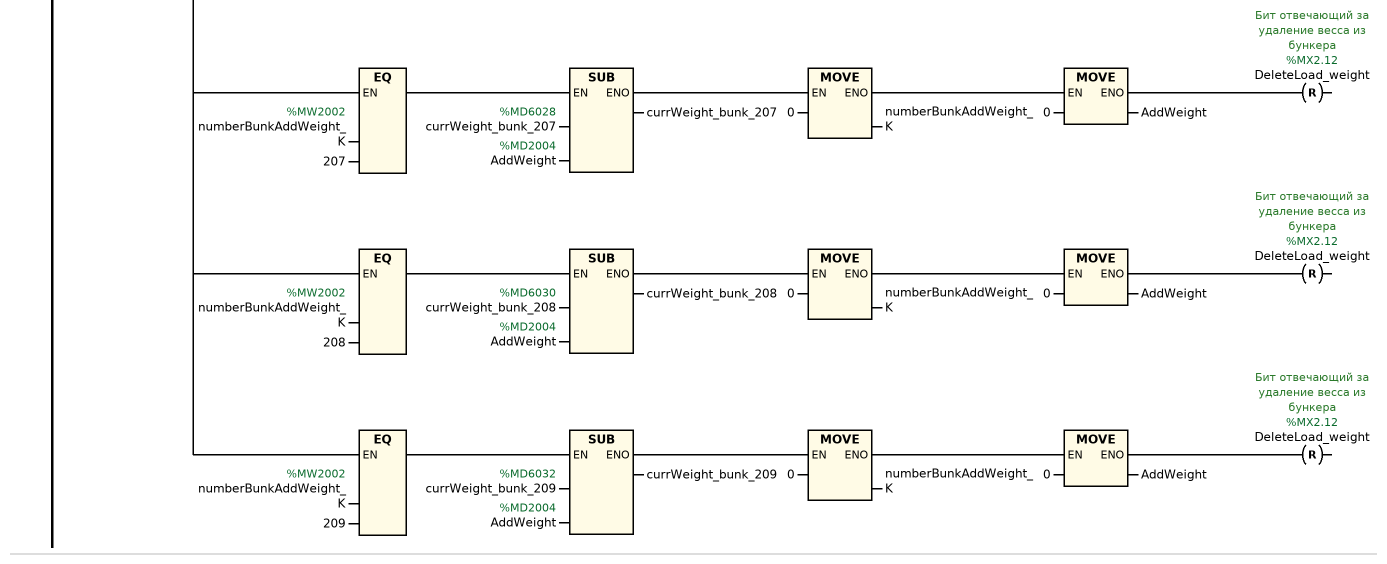
// NETWORK 2
//   DeleteLoad_weight: Бит отвечающий за удаление весса из бункера | AT %MX2.12
//   numberBunkAddWeight_Z: Храниться номер бункера для дабавления или удаления значения текущего весса в ручную... Сырье | AT %MW2000
//   currWeight_bunk_101: ----------------------------------------------------------------------------------------------------- текущий вес в зерновых бункерах ----------------------------------------------------------------------------------------------------- | AT %MD6000
//   AddWeight: Значение дабавляемого весса в бункер | AT %MD2004
//   currWeight_bunk_102: AT %MD6002
//   currWeight_bunk_103: AT %MD6004
//   currWeight_bunk_104: AT %MD6006
//   currWeight_bunk_105: AT %MD6008
//   currWeight_bunk_106: AT %MD6010
//   currWeight_bunk_107: AT %MD6012
//   currWeight_bunk_108: AT %MD6014
//   numberBunkAddWeight_K: Храниться номер бункера для дабавления или удаления значения текущего весса в ручную... Добавки | AT %MW2002
//   currWeight_bunk_201: ----------------------------------------------------------------------------------------------------- ----------------------------------------------------------------------------------------------------- текущий вес в бункерах компонентов ----------------------------------------------------------------------------------------------------- | AT %MD6016
//   currWeight_bunk_202: AT %MD6018
//   currWeight_bunk_203: AT %MD6020
//   currWeight_bunk_204: AT %MD6022
//   currWeight_bunk_205: AT %MD6024
//   currWeight_bunk_206: AT %MD6026
//   currWeight_bunk_207: AT %MD6028
//   currWeight_bunk_208: AT %MD6030
//   currWeight_bunk_209: AT %MD6032
_w2 := DeleteLoad_weight;
IF _w2 AND numberBunkAddWeight_Z = 101 THEN currWeight_bunk_101 := currWeight_bunk_101 - AddWeight; END_IF
IF _w2 AND numberBunkAddWeight_Z = 101 THEN numberBunkAddWeight_Z := 0; END_IF
IF _w2 AND numberBunkAddWeight_Z = 101 THEN AddWeight := 0; END_IF
DeleteLoad_weight R= _w2 AND numberBunkAddWeight_Z = 101;
IF _w2 AND numberBunkAddWeight_Z = 102 THEN currWeight_bunk_102 := currWeight_bunk_102 - AddWeight; END_IF
IF _w2 AND numberBunkAddWeight_Z = 102 THEN numberBunkAddWeight_Z := 0; END_IF
IF _w2 AND numberBunkAddWeight_Z = 102 THEN AddWeight := 0; END_IF
DeleteLoad_weight R= _w2 AND numberBunkAddWeight_Z = 102;
IF _w2 AND numberBunkAddWeight_Z = 103 THEN currWeight_bunk_103 := currWeight_bunk_103 - AddWeight; END_IF
IF _w2 AND numberBunkAddWeight_Z = 103 THEN numberBunkAddWeight_Z := 0; END_IF
IF _w2 AND numberBunkAddWeight_Z = 103 THEN AddWeight := 0; END_IF
DeleteLoad_weight R= _w2 AND numberBunkAddWeight_Z = 103;
IF _w2 AND numberBunkAddWeight_Z = 104 THEN currWeight_bunk_104 := currWeight_bunk_104 - AddWeight; END_IF
IF _w2 AND numberBunkAddWeight_Z = 104 THEN numberBunkAddWeight_Z := 0; END_IF
IF _w2 AND numberBunkAddWeight_Z = 104 THEN AddWeight := 0; END_IF
DeleteLoad_weight R= _w2 AND numberBunkAddWeight_Z = 104;
IF _w2 AND numberBunkAddWeight_Z = 105 THEN currWeight_bunk_105 := currWeight_bunk_105 - AddWeight; END_IF
IF _w2 AND numberBunkAddWeight_Z = 105 THEN numberBunkAddWeight_Z := 0; END_IF
IF _w2 AND numberBunkAddWeight_Z = 105 THEN AddWeight := 0; END_IF
DeleteLoad_weight R= _w2 AND numberBunkAddWeight_Z = 105;
IF _w2 AND numberBunkAddWeight_Z = 106 THEN currWeight_bunk_106 := currWeight_bunk_106 - AddWeight; END_IF
IF _w2 AND numberBunkAddWeight_Z = 106 THEN numberBunkAddWeight_Z := 0; END_IF
IF _w2 AND numberBunkAddWeight_Z = 106 THEN AddWeight := 0; END_IF
DeleteLoad_weight R= _w2 AND numberBunkAddWeight_Z = 106;
IF _w2 AND numberBunkAddWeight_Z = 107 THEN currWeight_bunk_107 := currWeight_bunk_107 - AddWeight; END_IF
IF _w2 AND numberBunkAddWeight_Z = 107 THEN numberBunkAddWeight_Z := 0; END_IF
IF _w2 AND numberBunkAddWeight_Z = 107 THEN AddWeight := 0; END_IF
DeleteLoad_weight R= _w2 AND numberBunkAddWeight_Z = 107;
IF _w2 AND numberBunkAddWeight_Z = 108 THEN currWeight_bunk_108 := currWeight_bunk_108 - AddWeight; END_IF
IF _w2 AND numberBunkAddWeight_Z = 108 THEN numberBunkAddWeight_Z := 0; END_IF
IF _w2 AND numberBunkAddWeight_Z = 108 THEN AddWeight := 0; END_IF
DeleteLoad_weight R= _w2 AND numberBunkAddWeight_Z = 108;
IF _w2 AND numberBunkAddWeight_K = 201 THEN currWeight_bunk_201 := currWeight_bunk_201 - AddWeight; END_IF
IF _w2 AND numberBunkAddWeight_K = 201 THEN numberBunkAddWeight_K := 0; END_IF
IF _w2 AND numberBunkAddWeight_K = 201 THEN AddWeight := 0; END_IF
DeleteLoad_weight R= _w2 AND numberBunkAddWeight_K = 201;
IF _w2 AND numberBunkAddWeight_K = 202 THEN currWeight_bunk_202 := currWeight_bunk_202 - AddWeight; END_IF
IF _w2 AND numberBunkAddWeight_K = 202 THEN numberBunkAddWeight_K := 0; END_IF
IF _w2 AND numberBunkAddWeight_K = 202 THEN AddWeight := 0; END_IF
DeleteLoad_weight R= _w2 AND numberBunkAddWeight_K = 202;
IF _w2 AND numberBunkAddWeight_K = 203 THEN currWeight_bunk_203 := currWeight_bunk_203 - AddWeight; END_IF
IF _w2 AND numberBunkAddWeight_K = 203 THEN numberBunkAddWeight_K := 0; END_IF
IF _w2 AND numberBunkAddWeight_K = 203 THEN AddWeight := 0; END_IF
DeleteLoad_weight R= _w2 AND numberBunkAddWeight_K = 203;
IF _w2 AND numberBunkAddWeight_K = 204 THEN currWeight_bunk_204 := currWeight_bunk_204 - AddWeight; END_IF
IF _w2 AND numberBunkAddWeight_K = 204 THEN numberBunkAddWeight_K := 0; END_IF
IF _w2 AND numberBunkAddWeight_K = 204 THEN AddWeight := 0; END_IF
DeleteLoad_weight R= _w2 AND numberBunkAddWeight_K = 204;
IF _w2 AND numberBunkAddWeight_K = 205 THEN currWeight_bunk_205 := currWeight_bunk_205 - AddWeight; END_IF
IF _w2 AND numberBunkAddWeight_K = 205 THEN numberBunkAddWeight_K := 0; END_IF
IF _w2 AND numberBunkAddWeight_K = 205 THEN AddWeight := 0; END_IF
DeleteLoad_weight R= _w2 AND numberBunkAddWeight_K = 205;
IF _w2 AND numberBunkAddWeight_K = 206 THEN currWeight_bunk_206 := currWeight_bunk_206 - AddWeight; END_IF
IF _w2 AND numberBunkAddWeight_K = 206 THEN numberBunkAddWeight_K := 0; END_IF
IF _w2 AND numberBunkAddWeight_K = 206 THEN AddWeight := 0; END_IF
DeleteLoad_weight R= _w2 AND numberBunkAddWeight_K = 206;
IF _w2 AND numberBunkAddWeight_K = 207 THEN currWeight_bunk_207 := currWeight_bunk_207 - AddWeight; END_IF
IF _w2 AND numberBunkAddWeight_K = 207 THEN numberBunkAddWeight_K := 0; END_IF
IF _w2 AND numberBunkAddWeight_K = 207 THEN AddWeight := 0; END_IF
DeleteLoad_weight R= _w2 AND numberBunkAddWeight_K = 207;
IF _w2 AND numberBunkAddWeight_K = 208 THEN currWeight_bunk_208 := currWeight_bunk_208 - AddWeight; END_IF
IF _w2 AND numberBunkAddWeight_K = 208 THEN numberBunkAddWeight_K := 0; END_IF
IF _w2 AND numberBunkAddWeight_K = 208 THEN AddWeight := 0; END_IF
DeleteLoad_weight R= _w2 AND numberBunkAddWeight_K = 208;
IF _w2 AND numberBunkAddWeight_K = 209 THEN currWeight_bunk_209 := currWeight_bunk_209 - AddWeight; END_IF
IF _w2 AND numberBunkAddWeight_K = 209 THEN numberBunkAddWeight_K := 0; END_IF
IF _w2 AND numberBunkAddWeight_K = 209 THEN AddWeight := 0; END_IF
DeleteLoad_weight R= _w2 AND numberBunkAddWeight_K = 209;

END_PROGRAM

// PLC_241/Application/CONVERT_REAL_TO_INT
PROGRAM CONVERT_REAL_TO_INT
VAR
END_VAR

								
								// Значение (процент компонента в рецепте)
	KP_101:= (INT_TO_REAL(iKP_101)/10.0);
	KP_102:= (INT_TO_REAL(iKP_102)/10.0);
	KP_103:= (INT_TO_REAL(iKP_103)/10.0);
	KP_104:= (INT_TO_REAL(iKP_104)/10.0);
	KP_105:= (INT_TO_REAL(iKP_105)/10.0);
	KP_106:= (INT_TO_REAL(iKP_106)/10.0);
	KP_107:= (INT_TO_REAL(iKP_107)/10.0);
	KP_108:= (INT_TO_REAL(iKP_108)/10.0);
	
								// Значение в кг, масса компонента в рецепте
	iK_101:= REAL_TO_INT(K_101*10.0);
	iK_102:= REAL_TO_INT(K_102*10.0);
	iK_103:= REAL_TO_INT(K_103*10.0);
	iK_104:= REAL_TO_INT(K_104*10.0);
	iK_105:= REAL_TO_INT(K_105*10.0);
	iK_106:= REAL_TO_INT(K_106*10.0);
	iK_107:= REAL_TO_INT(K_107*10.0);
	iK_108:= REAL_TO_INT(K_108*10.0);
	
								// Значение выбега 
	FALL_101:= (INT_TO_REAL(iFALL_101)/10.0);
	FALL_102:= (INT_TO_REAL(iFALL_102)/10.0);
	FALL_103:= (INT_TO_REAL(iFALL_103)/10.0);
	FALL_104:= (INT_TO_REAL(iFALL_104)/10.0);
	FALL_105:= (INT_TO_REAL(iFALL_105)/10.0);
	FALL_106:= (INT_TO_REAL(iFALL_106)/10.0);
	FALL_107:= (INT_TO_REAL(iFALL_107)/10.0);
	FALL_108:= (INT_TO_REAL(iFALL_108)/10.0);
	
								// Значение (Кг) при котором дазатор начинает снижать скорость дозирования для точного дозирования на весы
	vlDropSpeed_101:= (INT_TO_REAL(ivlDropSpeed_101)/10.0);
	vlDropSpeed_102:= (INT_TO_REAL(ivlDropSpeed_102)/10.0);
	vlDropSpeed_103:= (INT_TO_REAL(ivlDropSpeed_103)/10.0);
	vlDropSpeed_104:= (INT_TO_REAL(ivlDropSpeed_104)/10.0);
	vlDropSpeed_105:= (INT_TO_REAL(ivlDropSpeed_105)/10.0);
	vlDropSpeed_106:= (INT_TO_REAL(ivlDropSpeed_106)/10.0);
	vlDropSpeed_107:= (INT_TO_REAL(ivlDropSpeed_107)/10.0);
	vlDropSpeed_108:= (INT_TO_REAL(ivlDropSpeed_108)/10.0);
	
								// Значение (Кг) после автоматической коррекции падающег остоба (Выбега)
	iNewFall_101:= REAL_TO_INT(NewFall_101*10.0);
	iNewFall_102:= REAL_TO_INT(NewFall_102*10.0);
	iNewFall_103:= REAL_TO_INT(NewFall_103*10.0);
	iNewFall_104:= REAL_TO_INT(NewFall_104*10.0);
	iNewFall_105:= REAL_TO_INT(NewFall_105*10.0);
	iNewFall_106:= REAL_TO_INT(NewFall_106*10.0);
	iNewFall_107:= REAL_TO_INT(NewFall_107*10.0);
	iNewFall_108:= REAL_TO_INT(NewFall_108*10.0);

END_PROGRAM

// PLC_241/Application/POU/prgDOSING_BIG_WEIGHT
PROGRAM prgDOSING_BIG_WEIGHT
VAR
	Dozator_101: Dozator;
	T_20110: T;
	TON_pch_11_16: TON;
	
	vesi_big_done: BOOL;	// Вес сдозирован на весы
	Dozator_102: Dozator;
	Dozator_103: Dozator;
	Dozator_104: Dozator;
	Dozator_105: Dozator;
	Dozator_106: Dozator;
	TON_pch_17_18: TON;
	Dozator_107: Dozator;
	Dozator_108: Dozator;
	vesi_big_unldone: BOOL;
	TP_TARE_BIG: TP;
	CTU_BIG_WEIGHT: CTU;
END_VAR
VAR // added by the converter: edge detectors and wires of the graphical bodies
    _rt1, _rt2, _rt3, _rt4, _rt5, _rt6, _rt7, _rt8, _rt9, _rt10, _rt11 : R_TRIG;
    _ft1 : F_TRIG;
    _w1, _w2, _w3, _w4, _w5, _w6, _w7, _w8, _w9 : BOOL;
END_VAR

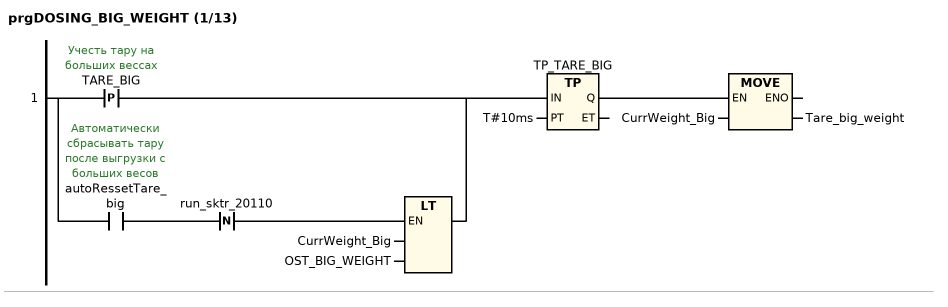
// NETWORK 1
//   TARE_BIG: Учесть тару на больших вессах
//   autoRessetTare_big: Автоматически сбрасывать тару после выгрузки с больших весов
//   CurrWeight_Big: Вес на больших весах
//   OST_BIG_WEIGHT: Остаток на больших весах (вводиться со скады)
//   Tare_big_weight: Вес тары на больших весах
_rt1(CLK := TARE_BIG);
_ft1(CLK := run_sktr_20110);
TP_TARE_BIG(IN := _rt1.Q OR autoRessetTare_big AND _ft1.Q AND CurrWeight_Big < OST_BIG_WEIGHT, PT := T#10ms); // TP
IF TP_TARE_BIG.Q THEN Tare_big_weight := CurrWeight_Big; END_IF

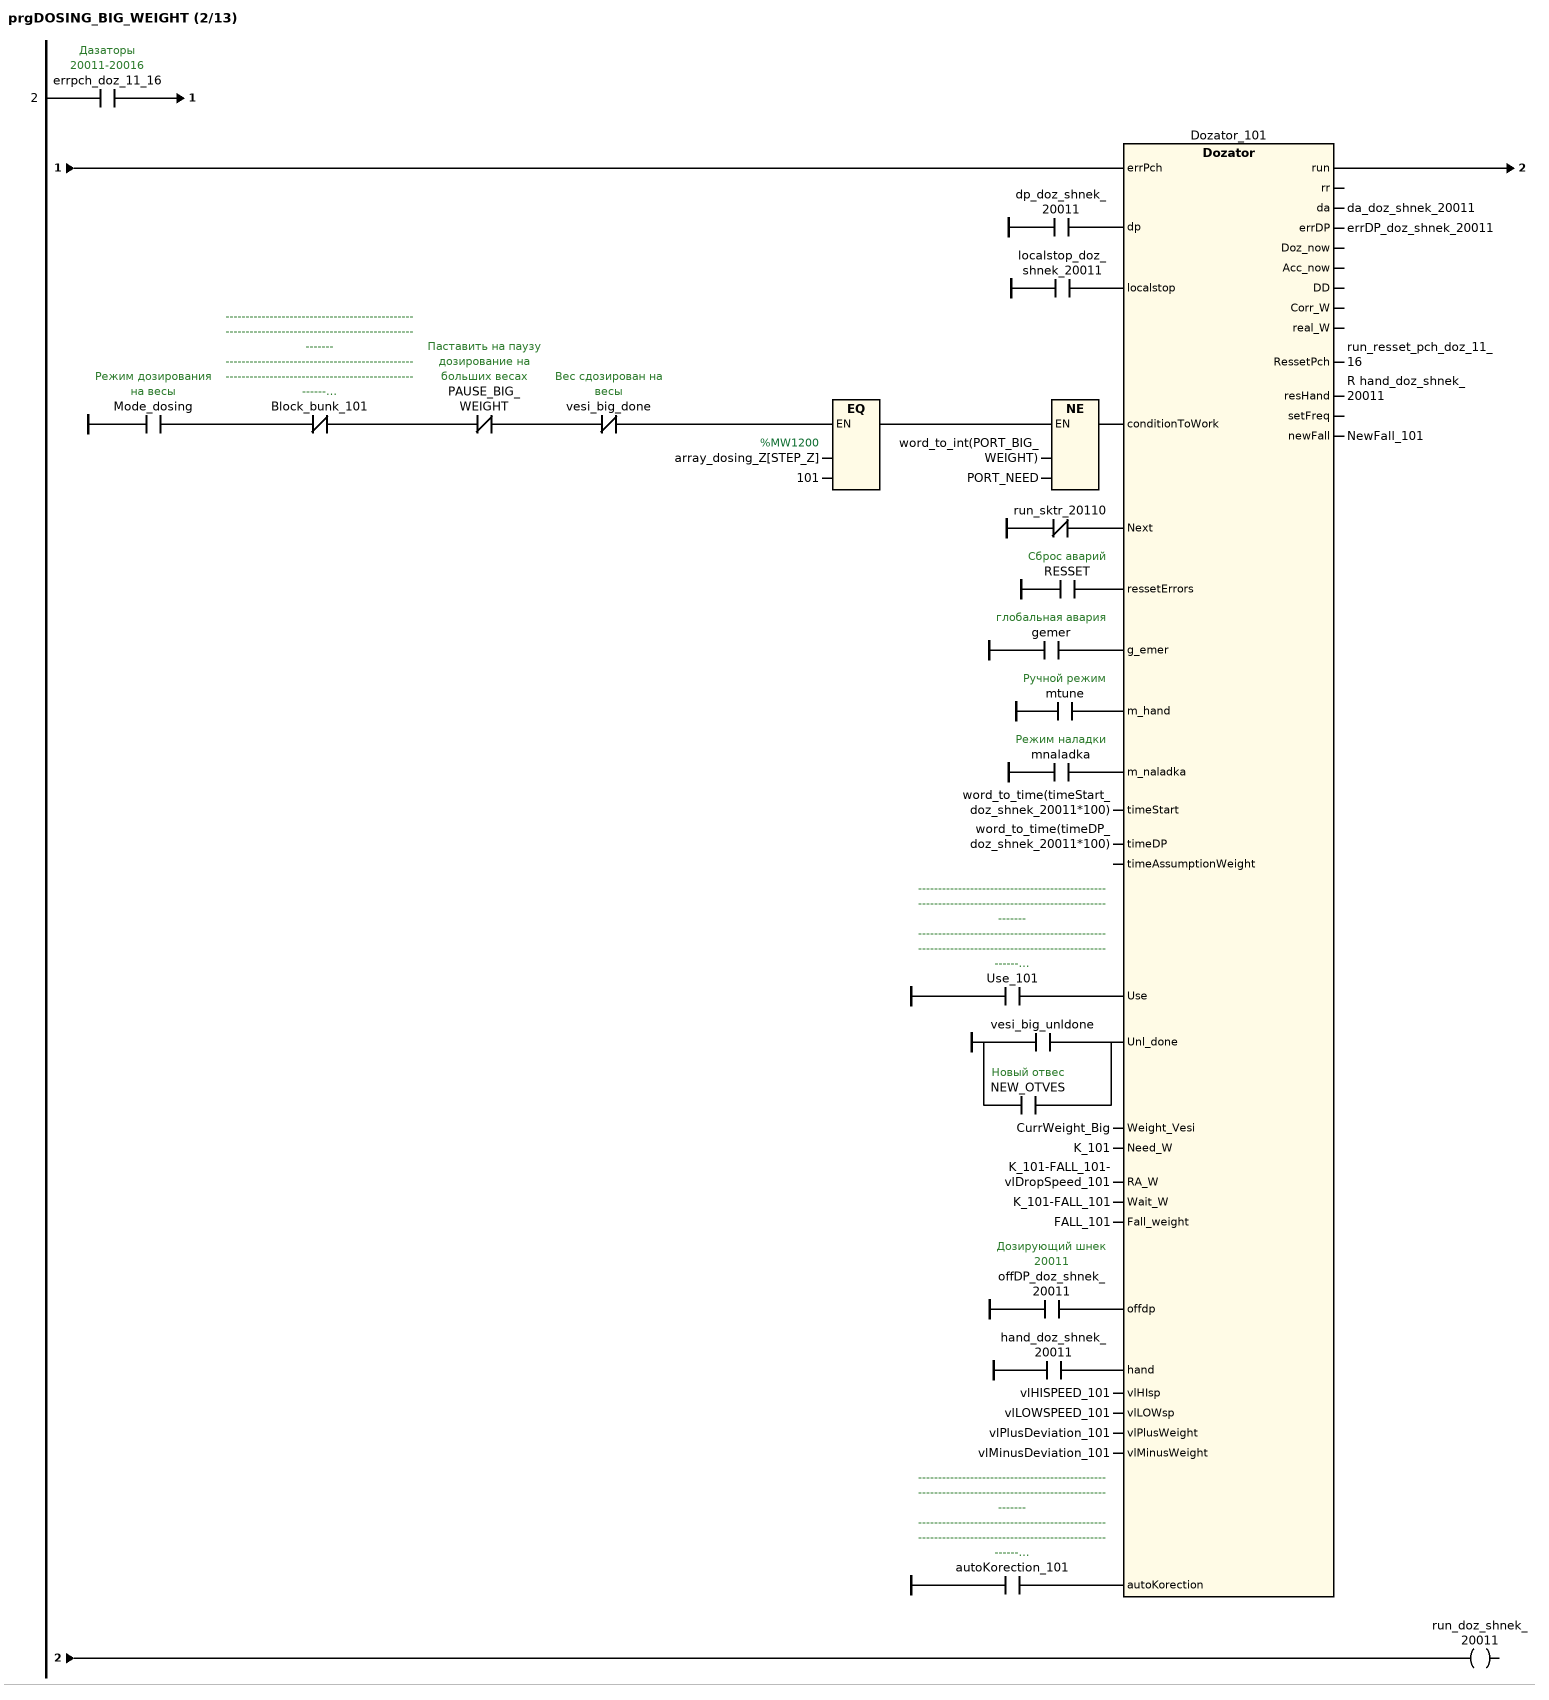
// NETWORK 2
//   errpch_doz_11_16: Дазаторы 20011-20016
//   Mode_dosing: Режим дозирования на весы
//   Block_bunk_101: ----------------------------------------------------------------------------------------------------- ----------------------------------------------------------------------------------------------------- Блокировка компонента на дозирование в рецепте -----------------------------------------------------------------------------------------------------
//   PAUSE_BIG_WEIGHT: Паставить на паузу дозирование на больших весах
//   vesi_big_done: Вес сдозирован на весы
//   array_dosing_Z[STEP_Z]: Массив очереди дозирования больших весов (в ячейке храниться номер бункера из которого нужно дозировать) | AT %MW1200
//   PORT_NEED: количество нужных порций
//   RESSET: Сброс аварий
//   gemer: глобальная авария
//   mtune: Ручной режим
//   mnaladka: Режим наладки
//   Use_101: ----------------------------------------------------------------------------------------------------- ----------------------------------------------------------------------------------------------------- Использование Дозатора в рецепте -----------------------------------------------------------------------------------------------------
//   NEW_OTVES: Новый отвес
//   CurrWeight_Big: Вес на больших весах
//   K_101: Значение реал для обработки контроллером
//   K_101-FALL_101-vlDropSpeed_101: Значение реал для обработки контроллером
//   K_101-FALL_101: Значение реал для обработки контроллером
//   FALL_101: Преобразованное значение падающего столба для обработки контроллером
//   offDP_doz_shnek_20011: Дозирующий шнек 20011
//   vlHISPEED_101: ----------------------------------------------------------------------------------------------------- ----------------------------------------------------------------------------------------------------- Значение (Гц) минимальной и максимальной скорости дозирования -----------------------------------------------------------------------------------------------------
//   vlPlusDeviation_101: ----------------------------------------------------------------------------------------------------- Значение (кг) допустимое отклонение +/- каждого компонента -----------------------------------------------------------------------------------------------------
//   autoKorection_101: ----------------------------------------------------------------------------------------------------- ----------------------------------------------------------------------------------------------------- Биты отвечающик за автоматический расчет падающего столба (Выбега) -----------------------------------------------------------------------------------------------------
//   errDP_doz_shnek_20011: Шнек Дозатор 20011
Dozator_101(
    errPch := errpch_doz_11_16,
    dp := dp_doz_shnek_20011,
    localstop := localstop_doz_shnek_20011,
    conditionToWork := Mode_dosing AND NOT Block_bunk_101 AND NOT PAUSE_BIG_WEIGHT AND NOT vesi_big_done AND array_dosing_Z[STEP_Z] = 101 AND (word_to_int(PORT_BIG_WEIGHT)) <> PORT_NEED,
    Next := NOT run_sktr_20110,
    ressetErrors := RESSET,
    g_emer := gemer,
    m_hand := mtune,
    m_naladka := mnaladka,
    timeStart := word_to_time(timeStart_doz_shnek_20011*100),
    timeDP := word_to_time(timeDP_doz_shnek_20011*100),
    Use := Use_101,
    Unl_done := vesi_big_unldone OR NEW_OTVES,
    Weight_Vesi := CurrWeight_Big,
    Need_W := K_101,
    RA_W := K_101-FALL_101-vlDropSpeed_101,
    Wait_W := K_101-FALL_101,
    Fall_weight := FALL_101,
    offdp := offDP_doz_shnek_20011,
    hand := hand_doz_shnek_20011,
    vlHIsp := vlHISPEED_101,
    vlLOWsp := vlLOWSPEED_101,
    vlPlusWeight := vlPlusDeviation_101,
    vlMinusWeight := vlMinusDeviation_101,
    autoKorection := autoKorection_101,
    da => da_doz_shnek_20011,
    errDP => errDP_doz_shnek_20011,
    RessetPch => run_resset_pch_doz_11_16,
    newFall => NewFall_101); // Dozator
hand_doz_shnek_20011 R= Dozator_101.resHand;
run_doz_shnek_20011 := Dozator_101.run;

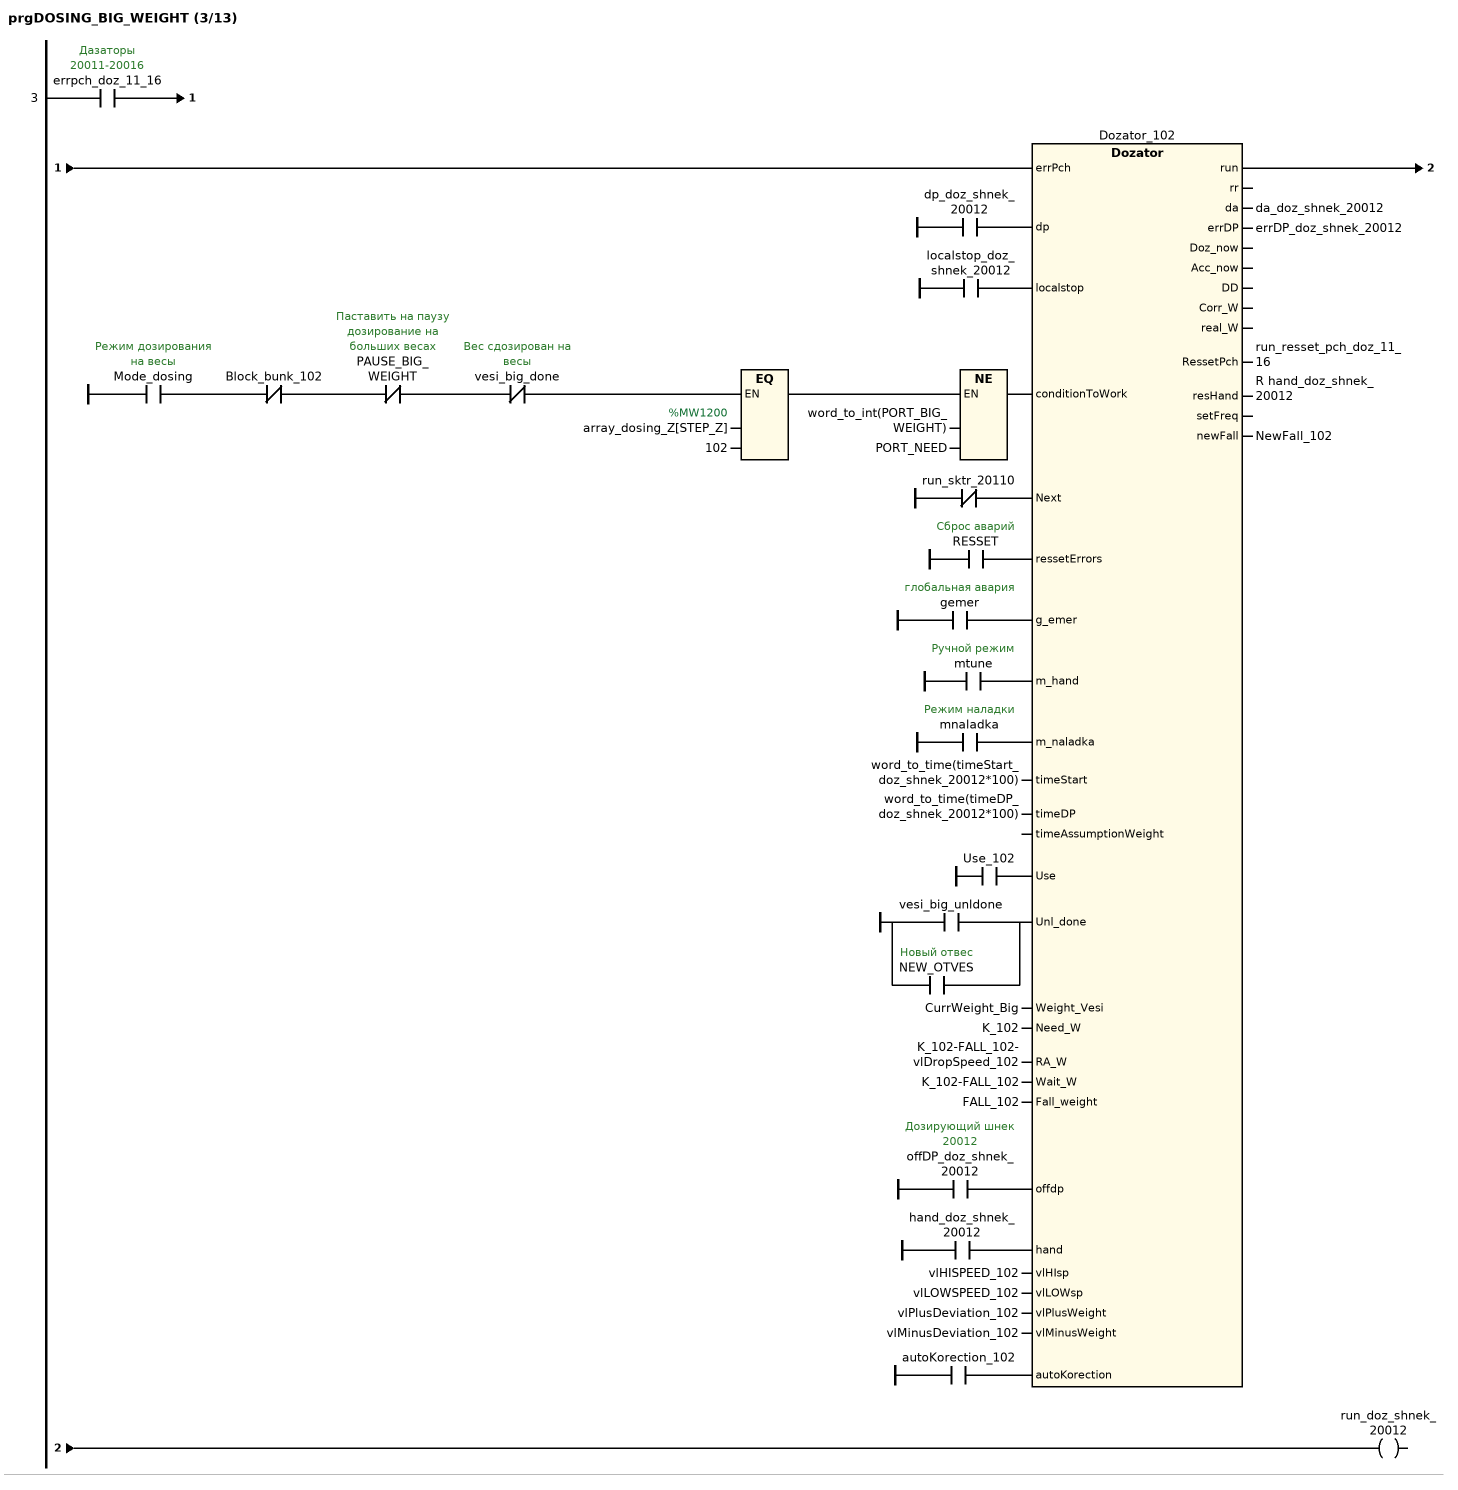
// NETWORK 3
//   errpch_doz_11_16: Дазаторы 20011-20016
//   Mode_dosing: Режим дозирования на весы
//   PAUSE_BIG_WEIGHT: Паставить на паузу дозирование на больших весах
//   vesi_big_done: Вес сдозирован на весы
//   array_dosing_Z[STEP_Z]: Массив очереди дозирования больших весов (в ячейке храниться номер бункера из которого нужно дозировать) | AT %MW1200
//   PORT_NEED: количество нужных порций
//   RESSET: Сброс аварий
//   gemer: глобальная авария
//   mtune: Ручной режим
//   mnaladka: Режим наладки
//   NEW_OTVES: Новый отвес
//   CurrWeight_Big: Вес на больших весах
//   offDP_doz_shnek_20012: Дозирующий шнек 20012
//   errDP_doz_shnek_20012: Шнек Дозатор 20012
Dozator_102(
    errPch := errpch_doz_11_16,
    dp := dp_doz_shnek_20012,
    localstop := localstop_doz_shnek_20012,
    conditionToWork := Mode_dosing AND NOT Block_bunk_102 AND NOT PAUSE_BIG_WEIGHT AND NOT vesi_big_done AND array_dosing_Z[STEP_Z] = 102 AND (word_to_int(PORT_BIG_WEIGHT)) <> PORT_NEED,
    Next := NOT run_sktr_20110,
    ressetErrors := RESSET,
    g_emer := gemer,
    m_hand := mtune,
    m_naladka := mnaladka,
    timeStart := word_to_time(timeStart_doz_shnek_20012*100),
    timeDP := word_to_time(timeDP_doz_shnek_20012*100),
    Use := Use_102,
    Unl_done := vesi_big_unldone OR NEW_OTVES,
    Weight_Vesi := CurrWeight_Big,
    Need_W := K_102,
    RA_W := K_102-FALL_102-vlDropSpeed_102,
    Wait_W := K_102-FALL_102,
    Fall_weight := FALL_102,
    offdp := offDP_doz_shnek_20012,
    hand := hand_doz_shnek_20012,
    vlHIsp := vlHISPEED_102,
    vlLOWsp := vlLOWSPEED_102,
    vlPlusWeight := vlPlusDeviation_102,
    vlMinusWeight := vlMinusDeviation_102,
    autoKorection := autoKorection_102,
    da => da_doz_shnek_20012,
    errDP => errDP_doz_shnek_20012,
    RessetPch => run_resset_pch_doz_11_16,
    newFall => NewFall_102); // Dozator
hand_doz_shnek_20012 R= Dozator_102.resHand;
run_doz_shnek_20012 := Dozator_102.run;

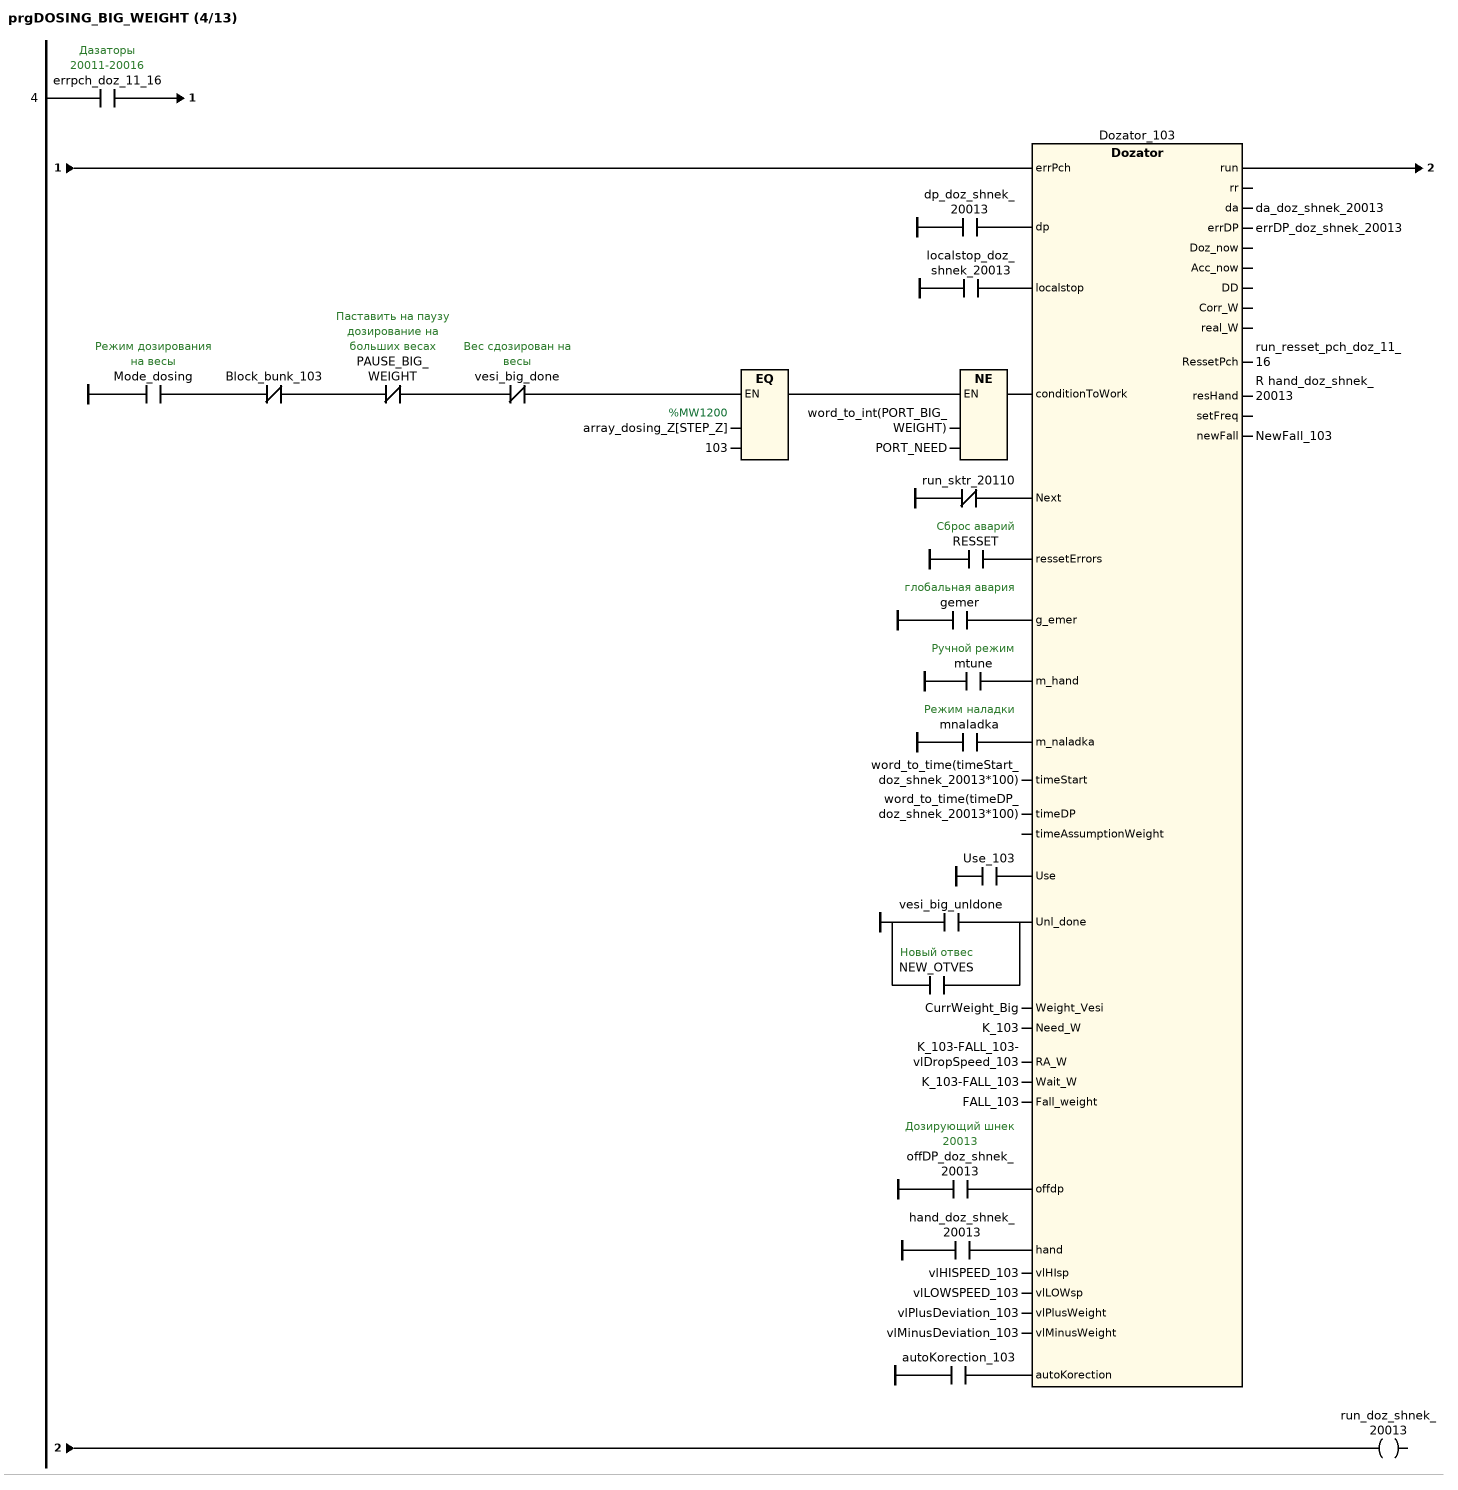
// NETWORK 4
//   errpch_doz_11_16: Дазаторы 20011-20016
//   Mode_dosing: Режим дозирования на весы
//   PAUSE_BIG_WEIGHT: Паставить на паузу дозирование на больших весах
//   vesi_big_done: Вес сдозирован на весы
//   array_dosing_Z[STEP_Z]: Массив очереди дозирования больших весов (в ячейке храниться номер бункера из которого нужно дозировать) | AT %MW1200
//   PORT_NEED: количество нужных порций
//   RESSET: Сброс аварий
//   gemer: глобальная авария
//   mtune: Ручной режим
//   mnaladka: Режим наладки
//   NEW_OTVES: Новый отвес
//   CurrWeight_Big: Вес на больших весах
//   offDP_doz_shnek_20013: Дозирующий шнек 20013
//   errDP_doz_shnek_20013: Шнек Дозатор 20013
Dozator_103(
    errPch := errpch_doz_11_16,
    dp := dp_doz_shnek_20013,
    localstop := localstop_doz_shnek_20013,
    conditionToWork := Mode_dosing AND NOT Block_bunk_103 AND NOT PAUSE_BIG_WEIGHT AND NOT vesi_big_done AND array_dosing_Z[STEP_Z] = 103 AND (word_to_int(PORT_BIG_WEIGHT)) <> PORT_NEED,
    Next := NOT run_sktr_20110,
    ressetErrors := RESSET,
    g_emer := gemer,
    m_hand := mtune,
    m_naladka := mnaladka,
    timeStart := word_to_time(timeStart_doz_shnek_20013*100),
    timeDP := word_to_time(timeDP_doz_shnek_20013*100),
    Use := Use_103,
    Unl_done := vesi_big_unldone OR NEW_OTVES,
    Weight_Vesi := CurrWeight_Big,
    Need_W := K_103,
    RA_W := K_103-FALL_103-vlDropSpeed_103,
    Wait_W := K_103-FALL_103,
    Fall_weight := FALL_103,
    offdp := offDP_doz_shnek_20013,
    hand := hand_doz_shnek_20013,
    vlHIsp := vlHISPEED_103,
    vlLOWsp := vlLOWSPEED_103,
    vlPlusWeight := vlPlusDeviation_103,
    vlMinusWeight := vlMinusDeviation_103,
    autoKorection := autoKorection_103,
    da => da_doz_shnek_20013,
    errDP => errDP_doz_shnek_20013,
    RessetPch => run_resset_pch_doz_11_16,
    newFall => NewFall_103); // Dozator
hand_doz_shnek_20013 R= Dozator_103.resHand;
run_doz_shnek_20013 := Dozator_103.run;

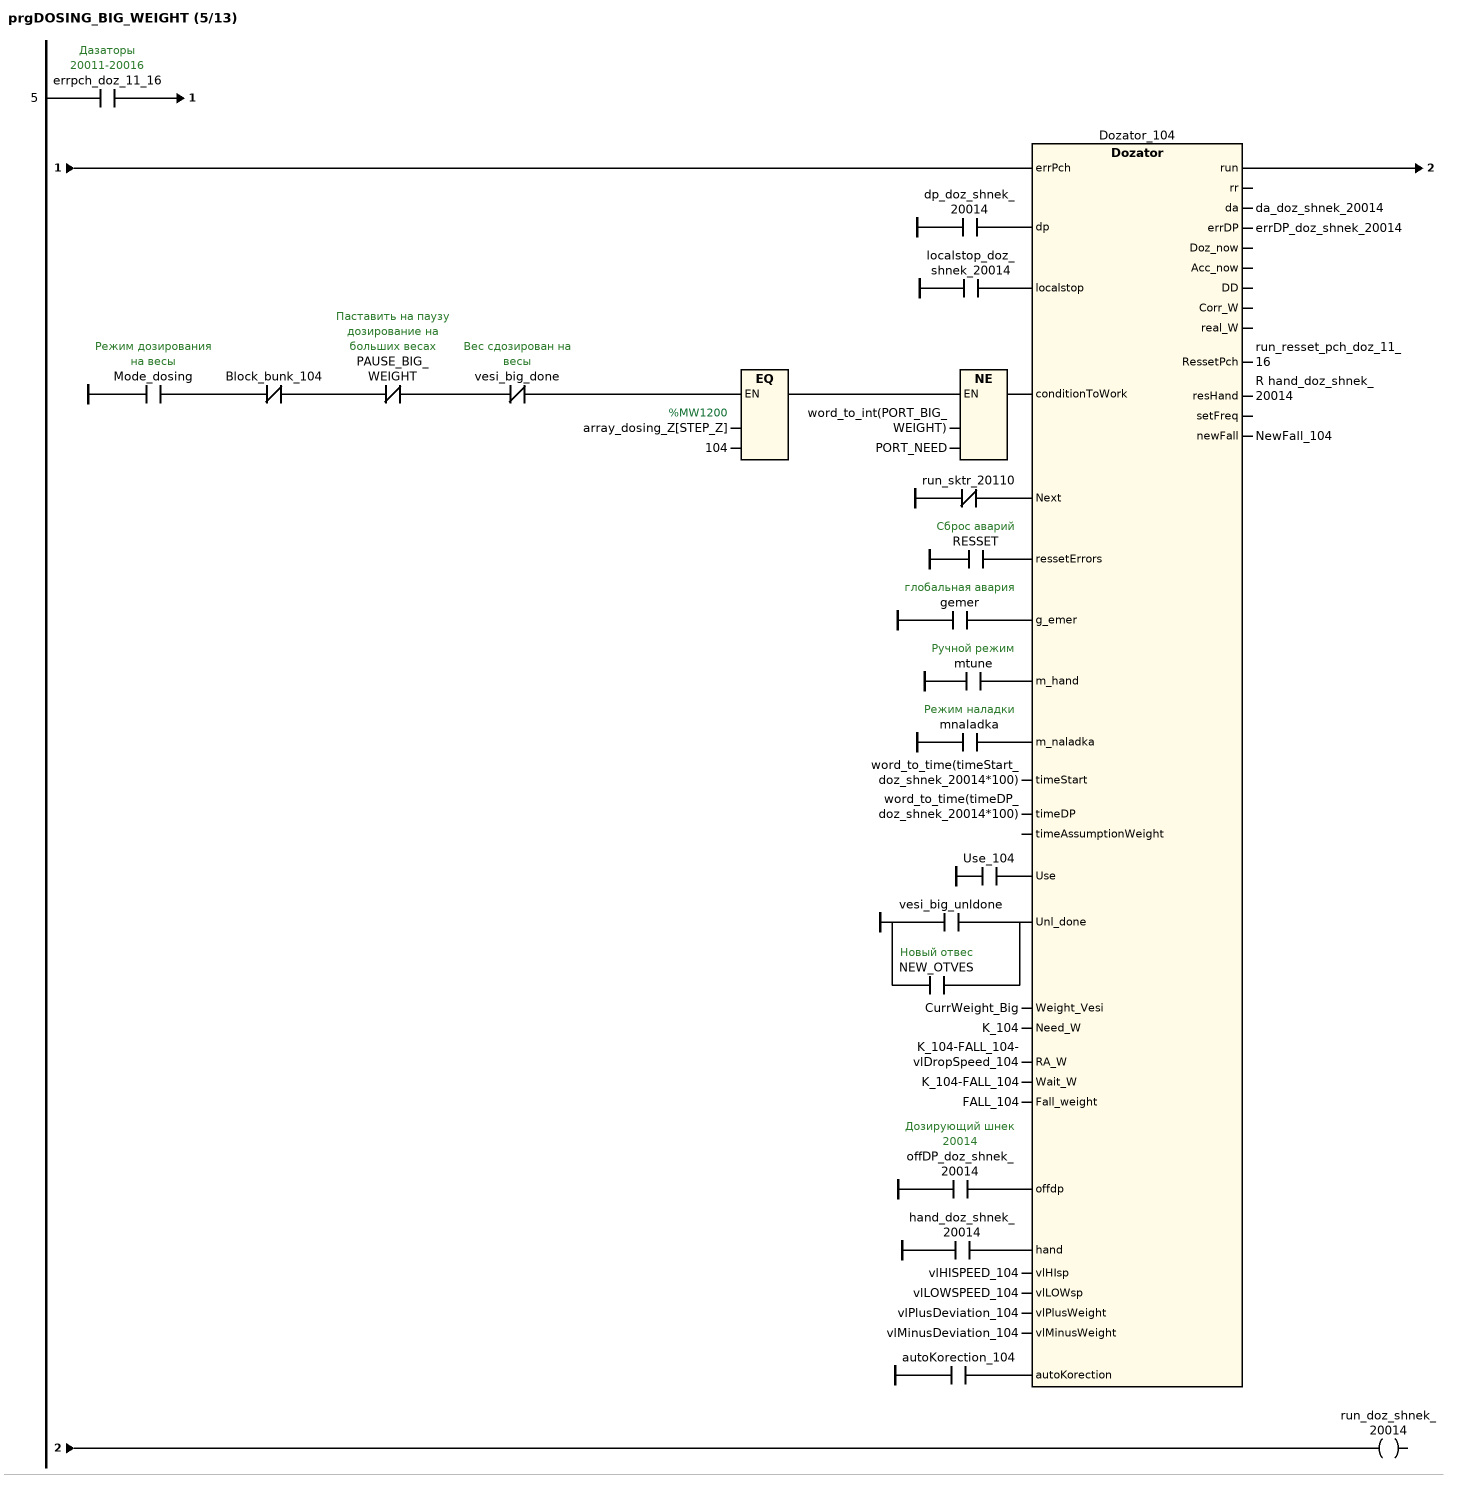
// NETWORK 5
//   errpch_doz_11_16: Дазаторы 20011-20016
//   Mode_dosing: Режим дозирования на весы
//   PAUSE_BIG_WEIGHT: Паставить на паузу дозирование на больших весах
//   vesi_big_done: Вес сдозирован на весы
//   array_dosing_Z[STEP_Z]: Массив очереди дозирования больших весов (в ячейке храниться номер бункера из которого нужно дозировать) | AT %MW1200
//   PORT_NEED: количество нужных порций
//   RESSET: Сброс аварий
//   gemer: глобальная авария
//   mtune: Ручной режим
//   mnaladka: Режим наладки
//   NEW_OTVES: Новый отвес
//   CurrWeight_Big: Вес на больших весах
//   offDP_doz_shnek_20014: Дозирующий шнек 20014
//   errDP_doz_shnek_20014: Шнек Дозатор 20014
Dozator_104(
    errPch := errpch_doz_11_16,
    dp := dp_doz_shnek_20014,
    localstop := localstop_doz_shnek_20014,
    conditionToWork := Mode_dosing AND NOT Block_bunk_104 AND NOT PAUSE_BIG_WEIGHT AND NOT vesi_big_done AND array_dosing_Z[STEP_Z] = 104 AND (word_to_int(PORT_BIG_WEIGHT)) <> PORT_NEED,
    Next := NOT run_sktr_20110,
    ressetErrors := RESSET,
    g_emer := gemer,
    m_hand := mtune,
    m_naladka := mnaladka,
    timeStart := word_to_time(timeStart_doz_shnek_20014*100),
    timeDP := word_to_time(timeDP_doz_shnek_20014*100),
    Use := Use_104,
    Unl_done := vesi_big_unldone OR NEW_OTVES,
    Weight_Vesi := CurrWeight_Big,
    Need_W := K_104,
    RA_W := K_104-FALL_104-vlDropSpeed_104,
    Wait_W := K_104-FALL_104,
    Fall_weight := FALL_104,
    offdp := offDP_doz_shnek_20014,
    hand := hand_doz_shnek_20014,
    vlHIsp := vlHISPEED_104,
    vlLOWsp := vlLOWSPEED_104,
    vlPlusWeight := vlPlusDeviation_104,
    vlMinusWeight := vlMinusDeviation_104,
    autoKorection := autoKorection_104,
    da => da_doz_shnek_20014,
    errDP => errDP_doz_shnek_20014,
    RessetPch => run_resset_pch_doz_11_16,
    newFall => NewFall_104); // Dozator
hand_doz_shnek_20014 R= Dozator_104.resHand;
run_doz_shnek_20014 := Dozator_104.run;

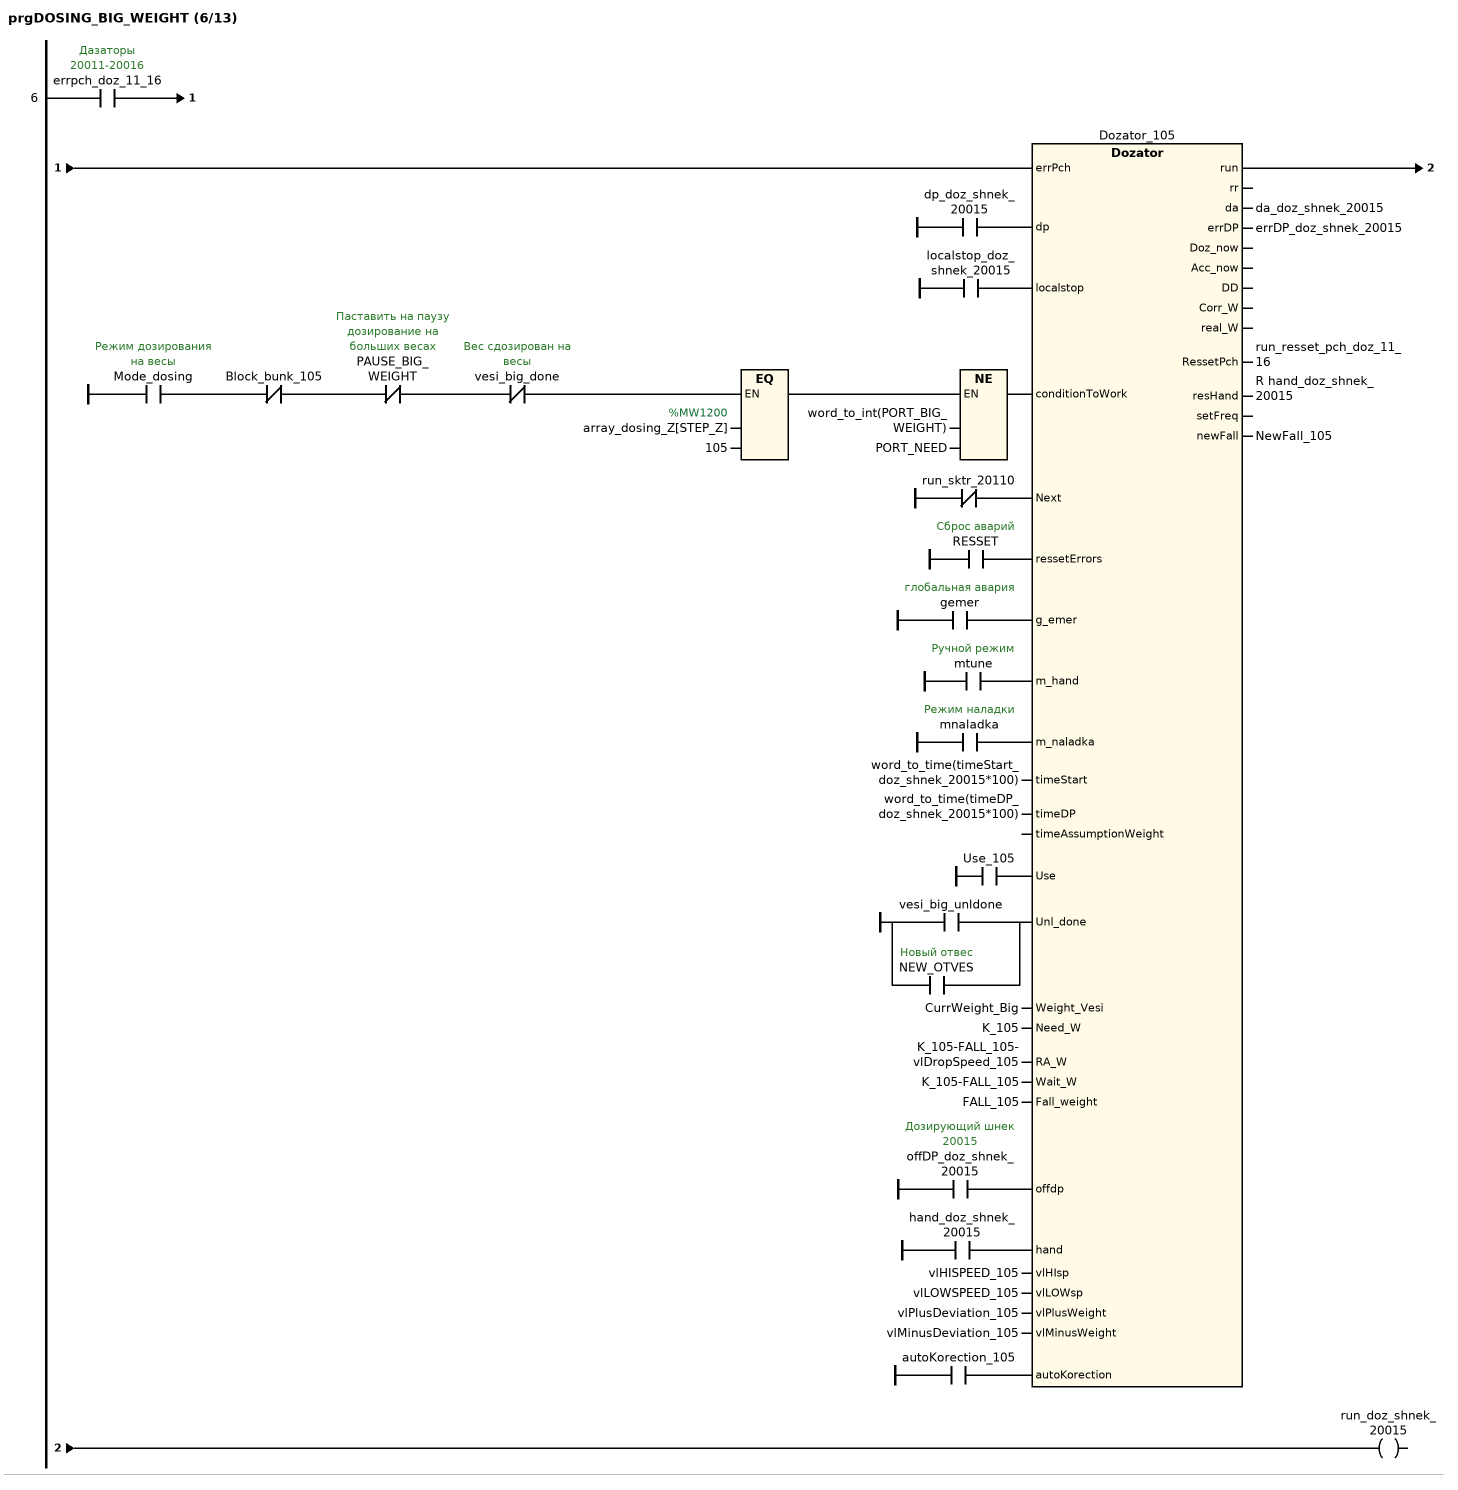
// NETWORK 6
//   errpch_doz_11_16: Дазаторы 20011-20016
//   Mode_dosing: Режим дозирования на весы
//   PAUSE_BIG_WEIGHT: Паставить на паузу дозирование на больших весах
//   vesi_big_done: Вес сдозирован на весы
//   array_dosing_Z[STEP_Z]: Массив очереди дозирования больших весов (в ячейке храниться номер бункера из которого нужно дозировать) | AT %MW1200
//   PORT_NEED: количество нужных порций
//   RESSET: Сброс аварий
//   gemer: глобальная авария
//   mtune: Ручной режим
//   mnaladka: Режим наладки
//   NEW_OTVES: Новый отвес
//   CurrWeight_Big: Вес на больших весах
//   offDP_doz_shnek_20015: Дозирующий шнек 20015
//   errDP_doz_shnek_20015: Шнек Дозатор 20015
Dozator_105(
    errPch := errpch_doz_11_16,
    dp := dp_doz_shnek_20015,
    localstop := localstop_doz_shnek_20015,
    conditionToWork := Mode_dosing AND NOT Block_bunk_105 AND NOT PAUSE_BIG_WEIGHT AND NOT vesi_big_done AND array_dosing_Z[STEP_Z] = 105 AND (word_to_int(PORT_BIG_WEIGHT)) <> PORT_NEED,
    Next := NOT run_sktr_20110,
    ressetErrors := RESSET,
    g_emer := gemer,
    m_hand := mtune,
    m_naladka := mnaladka,
    timeStart := word_to_time(timeStart_doz_shnek_20015*100),
    timeDP := word_to_time(timeDP_doz_shnek_20015*100),
    Use := Use_105,
    Unl_done := vesi_big_unldone OR NEW_OTVES,
    Weight_Vesi := CurrWeight_Big,
    Need_W := K_105,
    RA_W := K_105-FALL_105-vlDropSpeed_105,
    Wait_W := K_105-FALL_105,
    Fall_weight := FALL_105,
    offdp := offDP_doz_shnek_20015,
    hand := hand_doz_shnek_20015,
    vlHIsp := vlHISPEED_105,
    vlLOWsp := vlLOWSPEED_105,
    vlPlusWeight := vlPlusDeviation_105,
    vlMinusWeight := vlMinusDeviation_105,
    autoKorection := autoKorection_105,
    da => da_doz_shnek_20015,
    errDP => errDP_doz_shnek_20015,
    RessetPch => run_resset_pch_doz_11_16,
    newFall => NewFall_105); // Dozator
hand_doz_shnek_20015 R= Dozator_105.resHand;
run_doz_shnek_20015 := Dozator_105.run;

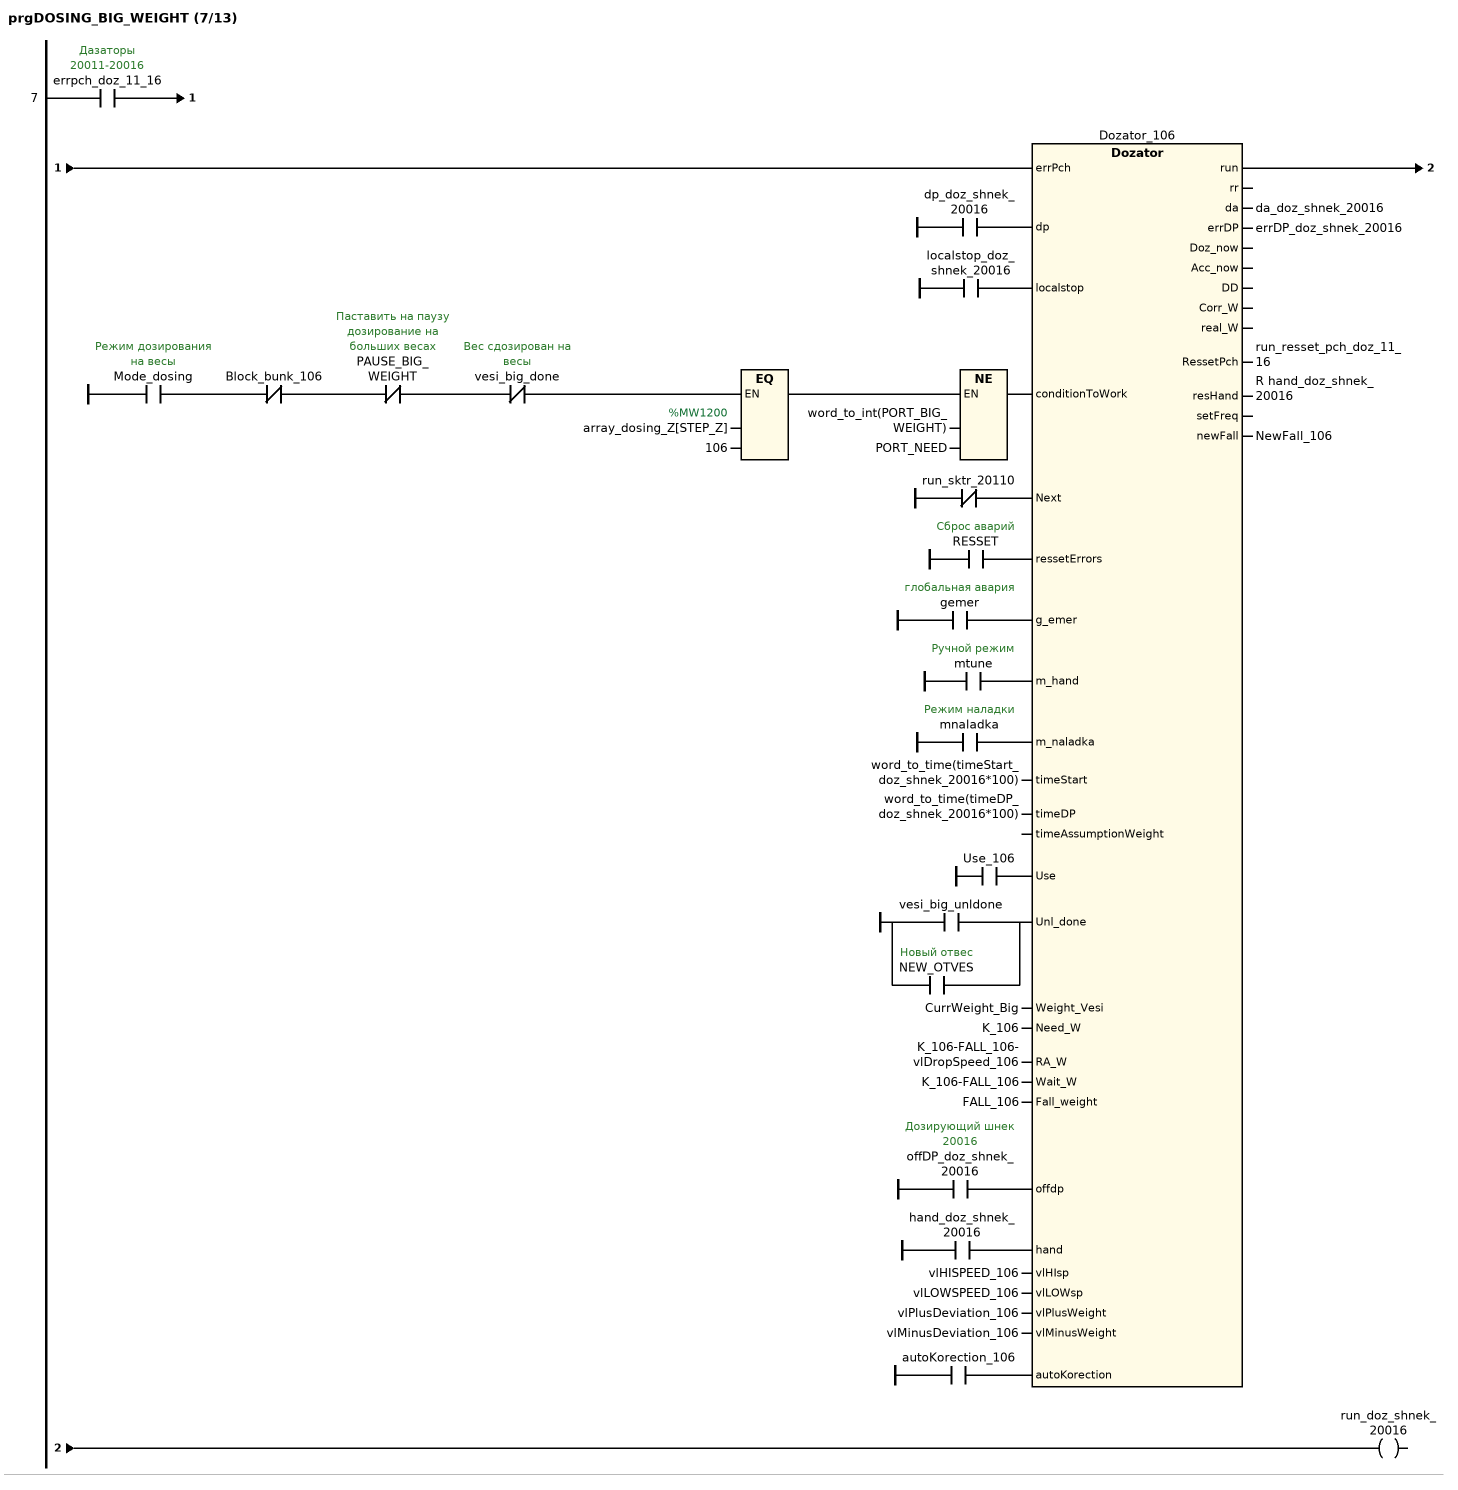
// NETWORK 7
//   errpch_doz_11_16: Дазаторы 20011-20016
//   Mode_dosing: Режим дозирования на весы
//   PAUSE_BIG_WEIGHT: Паставить на паузу дозирование на больших весах
//   vesi_big_done: Вес сдозирован на весы
//   array_dosing_Z[STEP_Z]: Массив очереди дозирования больших весов (в ячейке храниться номер бункера из которого нужно дозировать) | AT %MW1200
//   PORT_NEED: количество нужных порций
//   RESSET: Сброс аварий
//   gemer: глобальная авария
//   mtune: Ручной режим
//   mnaladka: Режим наладки
//   NEW_OTVES: Новый отвес
//   CurrWeight_Big: Вес на больших весах
//   offDP_doz_shnek_20016: Дозирующий шнек 20016
//   errDP_doz_shnek_20016: Шнек Дозатор 20016
Dozator_106(
    errPch := errpch_doz_11_16,
    dp := dp_doz_shnek_20016,
    localstop := localstop_doz_shnek_20016,
    conditionToWork := Mode_dosing AND NOT Block_bunk_106 AND NOT PAUSE_BIG_WEIGHT AND NOT vesi_big_done AND array_dosing_Z[STEP_Z] = 106 AND (word_to_int(PORT_BIG_WEIGHT)) <> PORT_NEED,
    Next := NOT run_sktr_20110,
    ressetErrors := RESSET,
    g_emer := gemer,
    m_hand := mtune,
    m_naladka := mnaladka,
    timeStart := word_to_time(timeStart_doz_shnek_20016*100),
    timeDP := word_to_time(timeDP_doz_shnek_20016*100),
    Use := Use_106,
    Unl_done := vesi_big_unldone OR NEW_OTVES,
    Weight_Vesi := CurrWeight_Big,
    Need_W := K_106,
    RA_W := K_106-FALL_106-vlDropSpeed_106,
    Wait_W := K_106-FALL_106,
    Fall_weight := FALL_106,
    offdp := offDP_doz_shnek_20016,
    hand := hand_doz_shnek_20016,
    vlHIsp := vlHISPEED_106,
    vlLOWsp := vlLOWSPEED_106,
    vlPlusWeight := vlPlusDeviation_106,
    vlMinusWeight := vlMinusDeviation_106,
    autoKorection := autoKorection_106,
    da => da_doz_shnek_20016,
    errDP => errDP_doz_shnek_20016,
    RessetPch => run_resset_pch_doz_11_16,
    newFall => NewFall_106); // Dozator
hand_doz_shnek_20016 R= Dozator_106.resHand;
run_doz_shnek_20016 := Dozator_106.run;

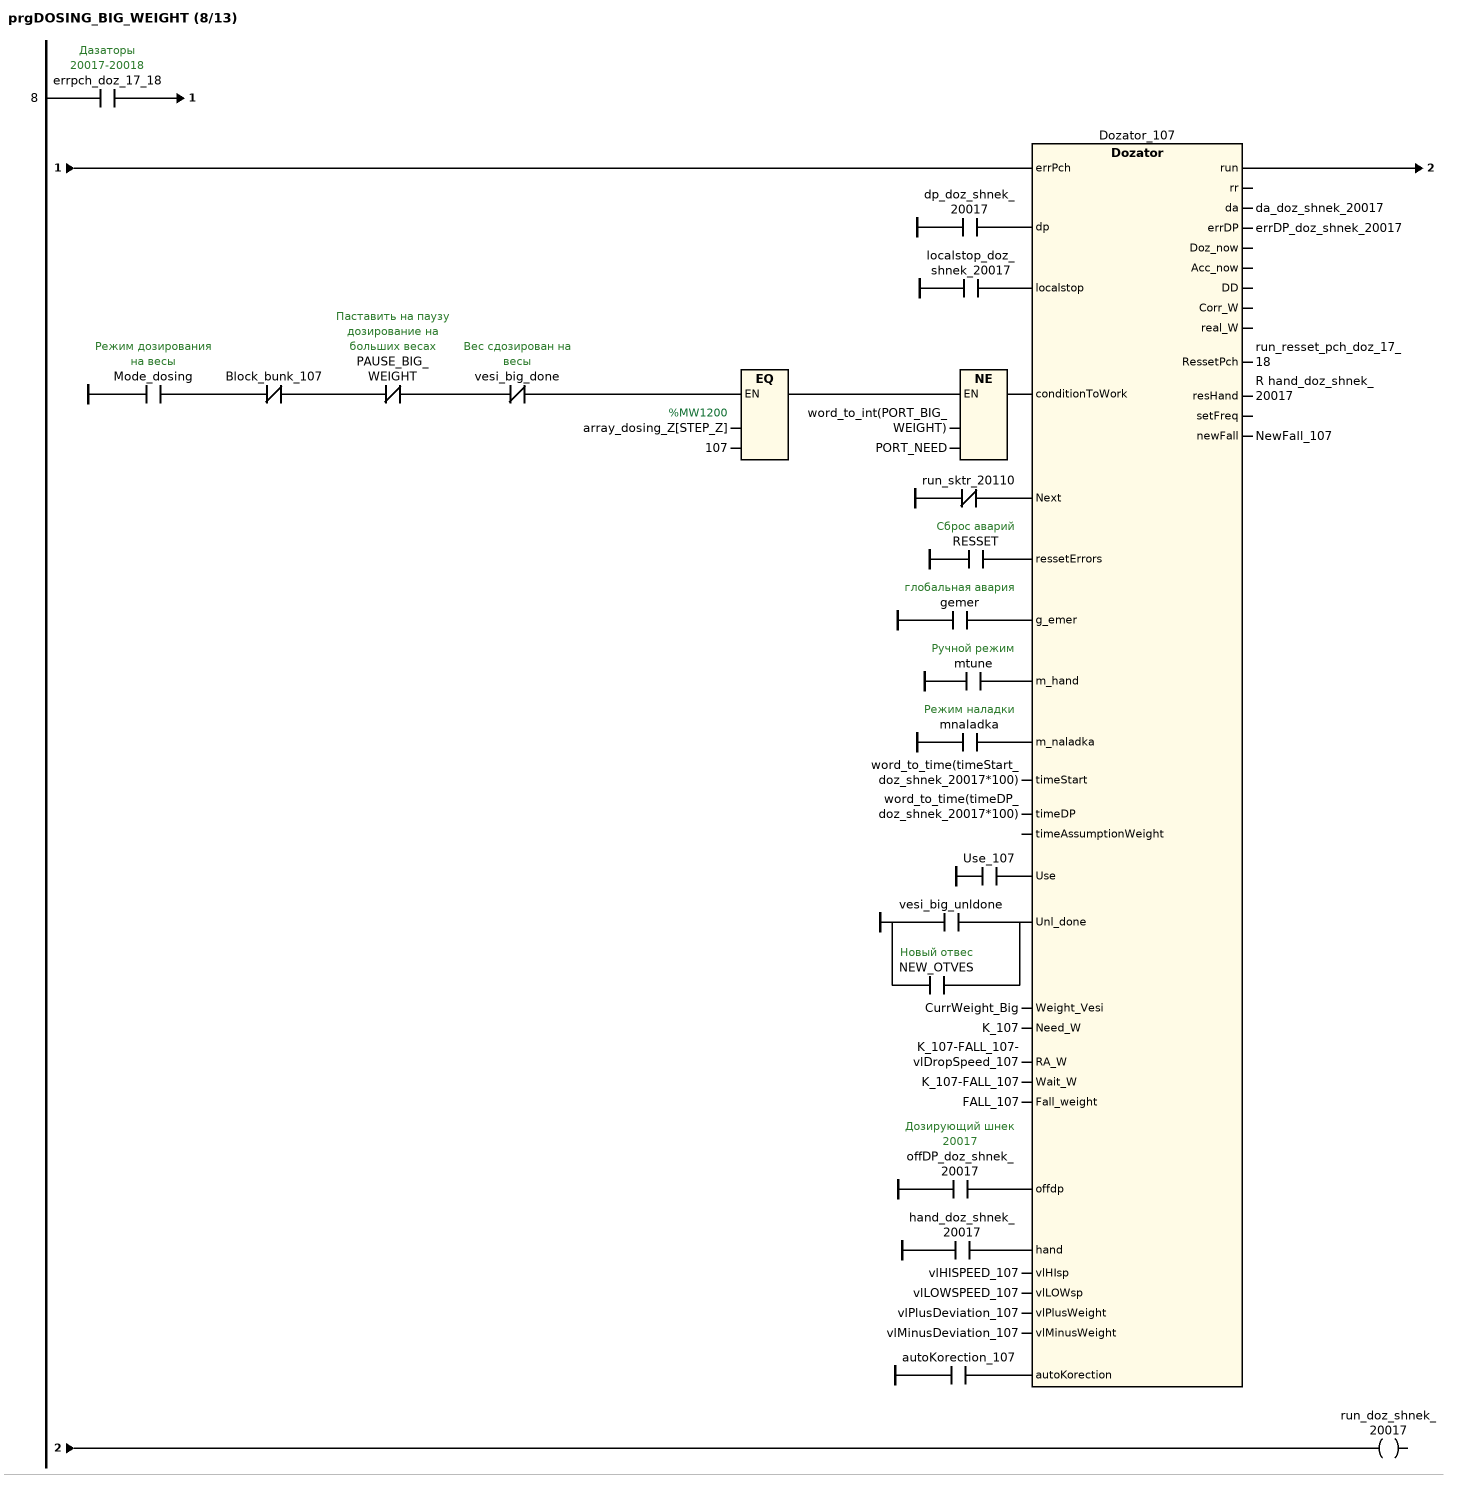
// NETWORK 8
//   errpch_doz_17_18: Дазаторы 20017-20018
//   Mode_dosing: Режим дозирования на весы
//   PAUSE_BIG_WEIGHT: Паставить на паузу дозирование на больших весах
//   vesi_big_done: Вес сдозирован на весы
//   array_dosing_Z[STEP_Z]: Массив очереди дозирования больших весов (в ячейке храниться номер бункера из которого нужно дозировать) | AT %MW1200
//   PORT_NEED: количество нужных порций
//   RESSET: Сброс аварий
//   gemer: глобальная авария
//   mtune: Ручной режим
//   mnaladka: Режим наладки
//   NEW_OTVES: Новый отвес
//   CurrWeight_Big: Вес на больших весах
//   offDP_doz_shnek_20017: Дозирующий шнек 20017
//   errDP_doz_shnek_20017: Шнек Дозатор 20017
Dozator_107(
    errPch := errpch_doz_17_18,
    dp := dp_doz_shnek_20017,
    localstop := localstop_doz_shnek_20017,
    conditionToWork := Mode_dosing AND NOT Block_bunk_107 AND NOT PAUSE_BIG_WEIGHT AND NOT vesi_big_done AND array_dosing_Z[STEP_Z] = 107 AND (word_to_int(PORT_BIG_WEIGHT)) <> PORT_NEED,
    Next := NOT run_sktr_20110,
    ressetErrors := RESSET,
    g_emer := gemer,
    m_hand := mtune,
    m_naladka := mnaladka,
    timeStart := word_to_time(timeStart_doz_shnek_20017*100),
    timeDP := word_to_time(timeDP_doz_shnek_20017*100),
    Use := Use_107,
    Unl_done := vesi_big_unldone OR NEW_OTVES,
    Weight_Vesi := CurrWeight_Big,
    Need_W := K_107,
    RA_W := K_107-FALL_107-vlDropSpeed_107,
    Wait_W := K_107-FALL_107,
    Fall_weight := FALL_107,
    offdp := offDP_doz_shnek_20017,
    hand := hand_doz_shnek_20017,
    vlHIsp := vlHISPEED_107,
    vlLOWsp := vlLOWSPEED_107,
    vlPlusWeight := vlPlusDeviation_107,
    vlMinusWeight := vlMinusDeviation_107,
    autoKorection := autoKorection_107,
    da => da_doz_shnek_20017,
    errDP => errDP_doz_shnek_20017,
    RessetPch => run_resset_pch_doz_17_18,
    newFall => NewFall_107); // Dozator
hand_doz_shnek_20017 R= Dozator_107.resHand;
run_doz_shnek_20017 := Dozator_107.run;

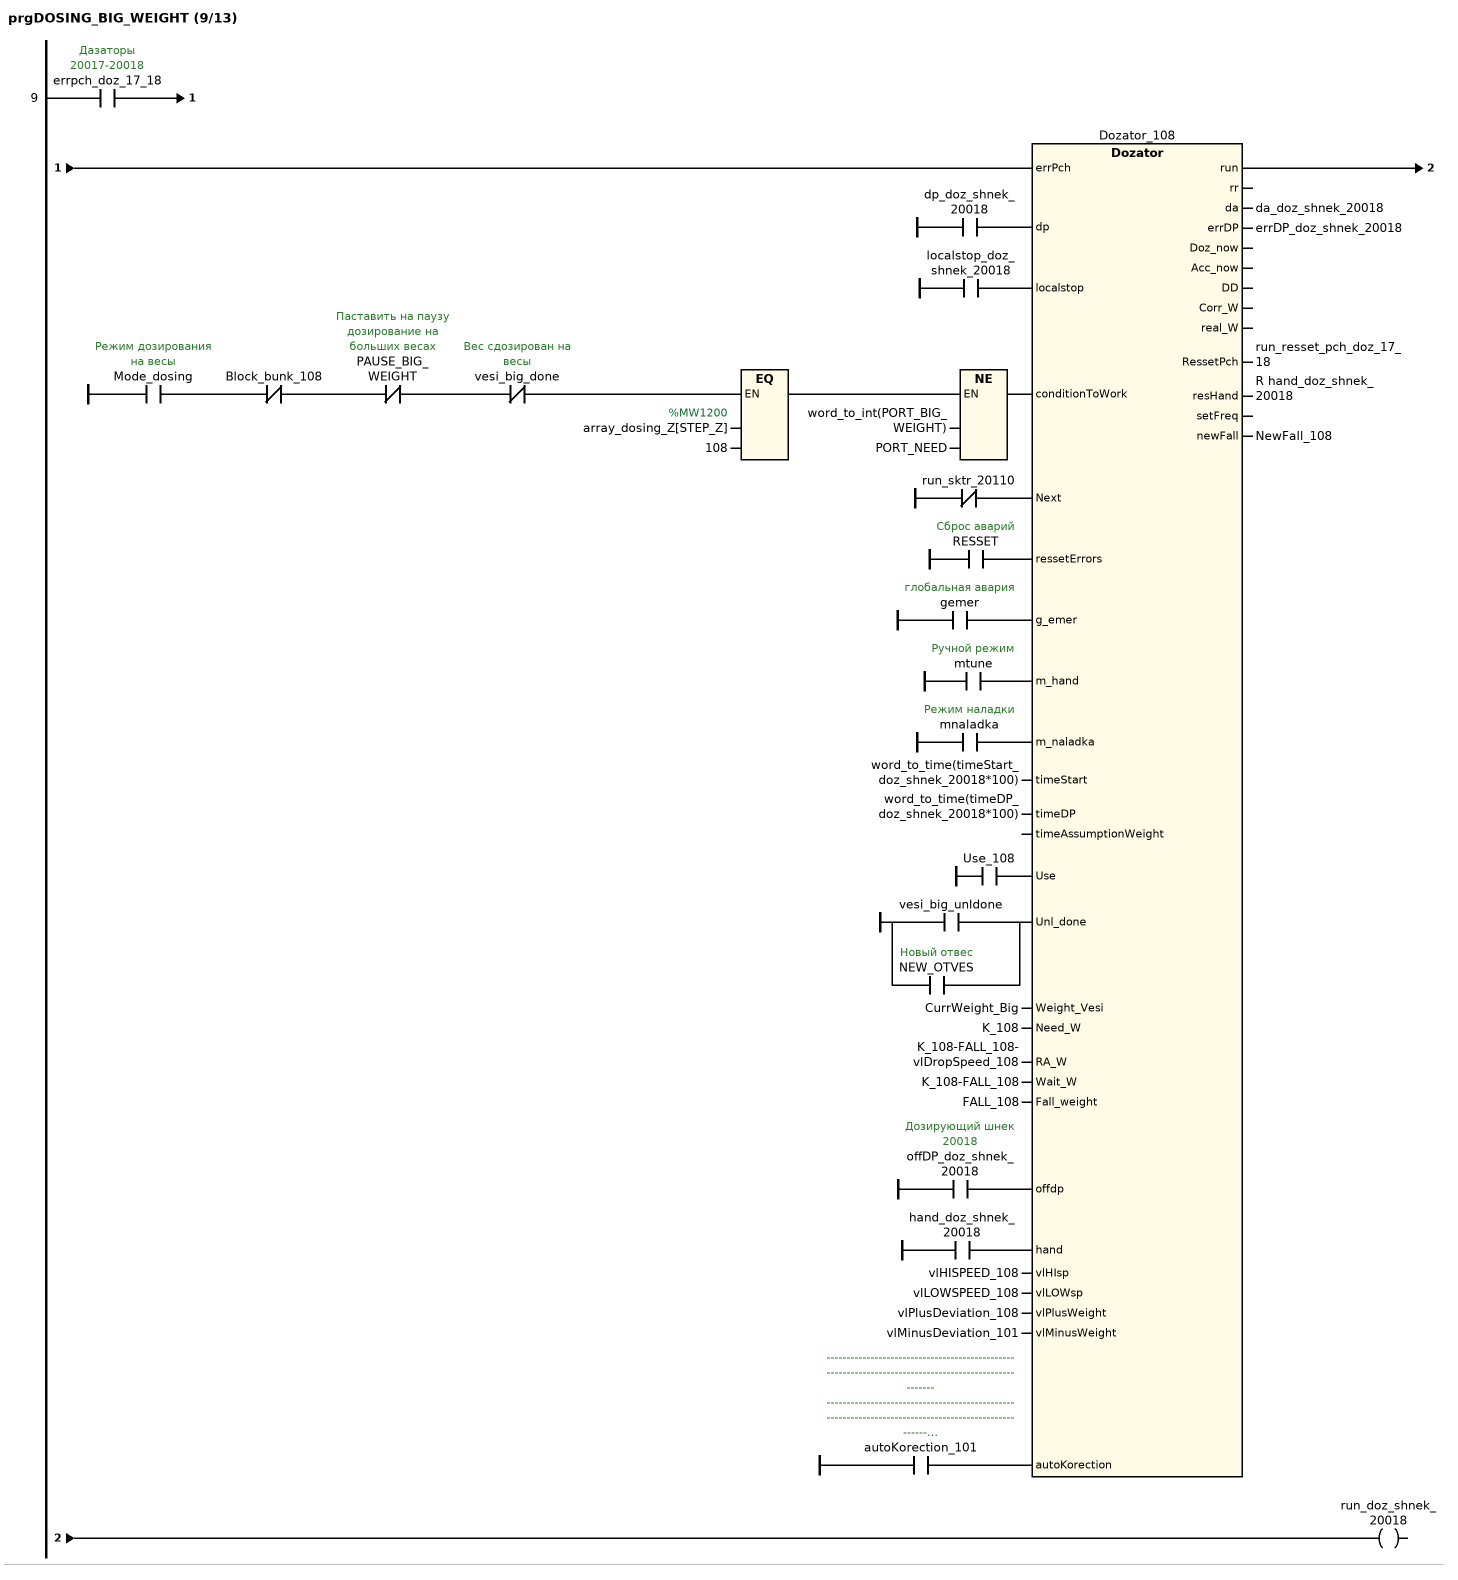
// NETWORK 9
//   errpch_doz_17_18: Дазаторы 20017-20018
//   Mode_dosing: Режим дозирования на весы
//   PAUSE_BIG_WEIGHT: Паставить на паузу дозирование на больших весах
//   vesi_big_done: Вес сдозирован на весы
//   array_dosing_Z[STEP_Z]: Массив очереди дозирования больших весов (в ячейке храниться номер бункера из которого нужно дозировать) | AT %MW1200
//   PORT_NEED: количество нужных порций
//   RESSET: Сброс аварий
//   gemer: глобальная авария
//   mtune: Ручной режим
//   mnaladka: Режим наладки
//   NEW_OTVES: Новый отвес
//   CurrWeight_Big: Вес на больших весах
//   offDP_doz_shnek_20018: Дозирующий шнек 20018
//   autoKorection_101: ----------------------------------------------------------------------------------------------------- ----------------------------------------------------------------------------------------------------- Биты отвечающик за автоматический расчет падающего столба (Выбега) -----------------------------------------------------------------------------------------------------
//   errDP_doz_shnek_20018: Шнек Дозатор 20018
Dozator_108(
    errPch := errpch_doz_17_18,
    dp := dp_doz_shnek_20018,
    localstop := localstop_doz_shnek_20018,
    conditionToWork := Mode_dosing AND NOT Block_bunk_108 AND NOT PAUSE_BIG_WEIGHT AND NOT vesi_big_done AND array_dosing_Z[STEP_Z] = 108 AND (word_to_int(PORT_BIG_WEIGHT)) <> PORT_NEED,
    Next := NOT run_sktr_20110,
    ressetErrors := RESSET,
    g_emer := gemer,
    m_hand := mtune,
    m_naladka := mnaladka,
    timeStart := word_to_time(timeStart_doz_shnek_20018*100),
    timeDP := word_to_time(timeDP_doz_shnek_20018*100),
    Use := Use_108,
    Unl_done := vesi_big_unldone OR NEW_OTVES,
    Weight_Vesi := CurrWeight_Big,
    Need_W := K_108,
    RA_W := K_108-FALL_108-vlDropSpeed_108,
    Wait_W := K_108-FALL_108,
    Fall_weight := FALL_108,
    offdp := offDP_doz_shnek_20018,
    hand := hand_doz_shnek_20018,
    vlHIsp := vlHISPEED_108,
    vlLOWsp := vlLOWSPEED_108,
    vlPlusWeight := vlPlusDeviation_108,
    vlMinusWeight := vlMinusDeviation_101,
    autoKorection := autoKorection_101,
    da => da_doz_shnek_20018,
    errDP => errDP_doz_shnek_20018,
    RessetPch => run_resset_pch_doz_17_18,
    newFall => NewFall_108); // Dozator
hand_doz_shnek_20018 R= Dozator_108.resHand;
run_doz_shnek_20018 := Dozator_108.run;

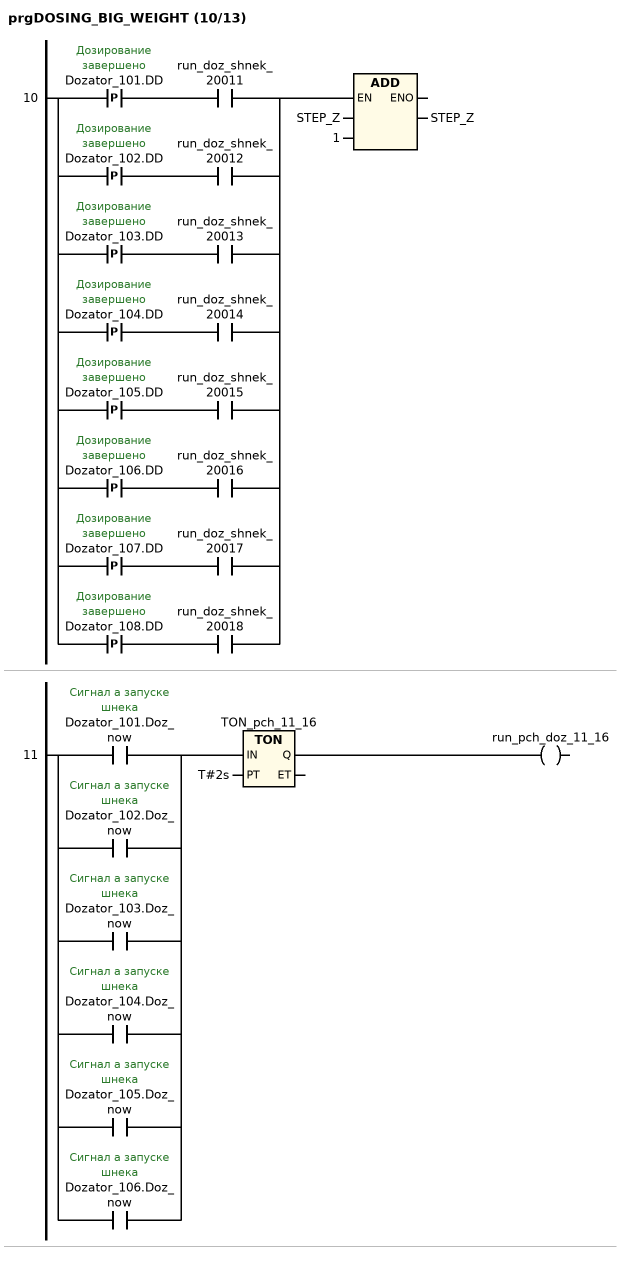
// NETWORK 10
//   Dozator_101.DD: Дозирование завершено
//   Dozator_102.DD: Дозирование завершено
//   Dozator_103.DD: Дозирование завершено
//   Dozator_104.DD: Дозирование завершено
//   Dozator_105.DD: Дозирование завершено
//   Dozator_106.DD: Дозирование завершено
//   Dozator_107.DD: Дозирование завершено
//   Dozator_108.DD: Дозирование завершено
//   STEP_Z: Стетчик для массива очереди дозирования больших вессов
_rt2(CLK := Dozator_101.DD);
_rt3(CLK := Dozator_102.DD);
_rt4(CLK := Dozator_103.DD);
_rt5(CLK := Dozator_104.DD);
_rt6(CLK := Dozator_105.DD);
_rt7(CLK := Dozator_106.DD);
_rt8(CLK := Dozator_107.DD);
_rt9(CLK := Dozator_108.DD);
IF _rt2.Q AND run_doz_shnek_20011 OR _rt3.Q AND run_doz_shnek_20012 OR _rt4.Q AND run_doz_shnek_20013 OR _rt5.Q AND run_doz_shnek_20014 OR _rt6.Q AND run_doz_shnek_20015 OR _rt7.Q AND run_doz_shnek_20016 OR _rt8.Q AND run_doz_shnek_20017 OR _rt9.Q AND run_doz_shnek_20018 THEN
    STEP_Z := STEP_Z + 1;
END_IF

// NETWORK 11
//   Dozator_101.Doz_now: Сигнал а запуске шнека
//   Dozator_102.Doz_now: Сигнал а запуске шнека
//   Dozator_103.Doz_now: Сигнал а запуске шнека
//   Dozator_104.Doz_now: Сигнал а запуске шнека
//   Dozator_105.Doz_now: Сигнал а запуске шнека
//   Dozator_106.Doz_now: Сигнал а запуске шнека
TON_pch_11_16(IN := Dozator_101.Doz_now OR Dozator_102.Doz_now OR Dozator_103.Doz_now OR Dozator_104.Doz_now OR Dozator_105.Doz_now OR Dozator_106.Doz_now, PT := T#2s); // TON
run_pch_doz_11_16 := TON_pch_11_16.Q;

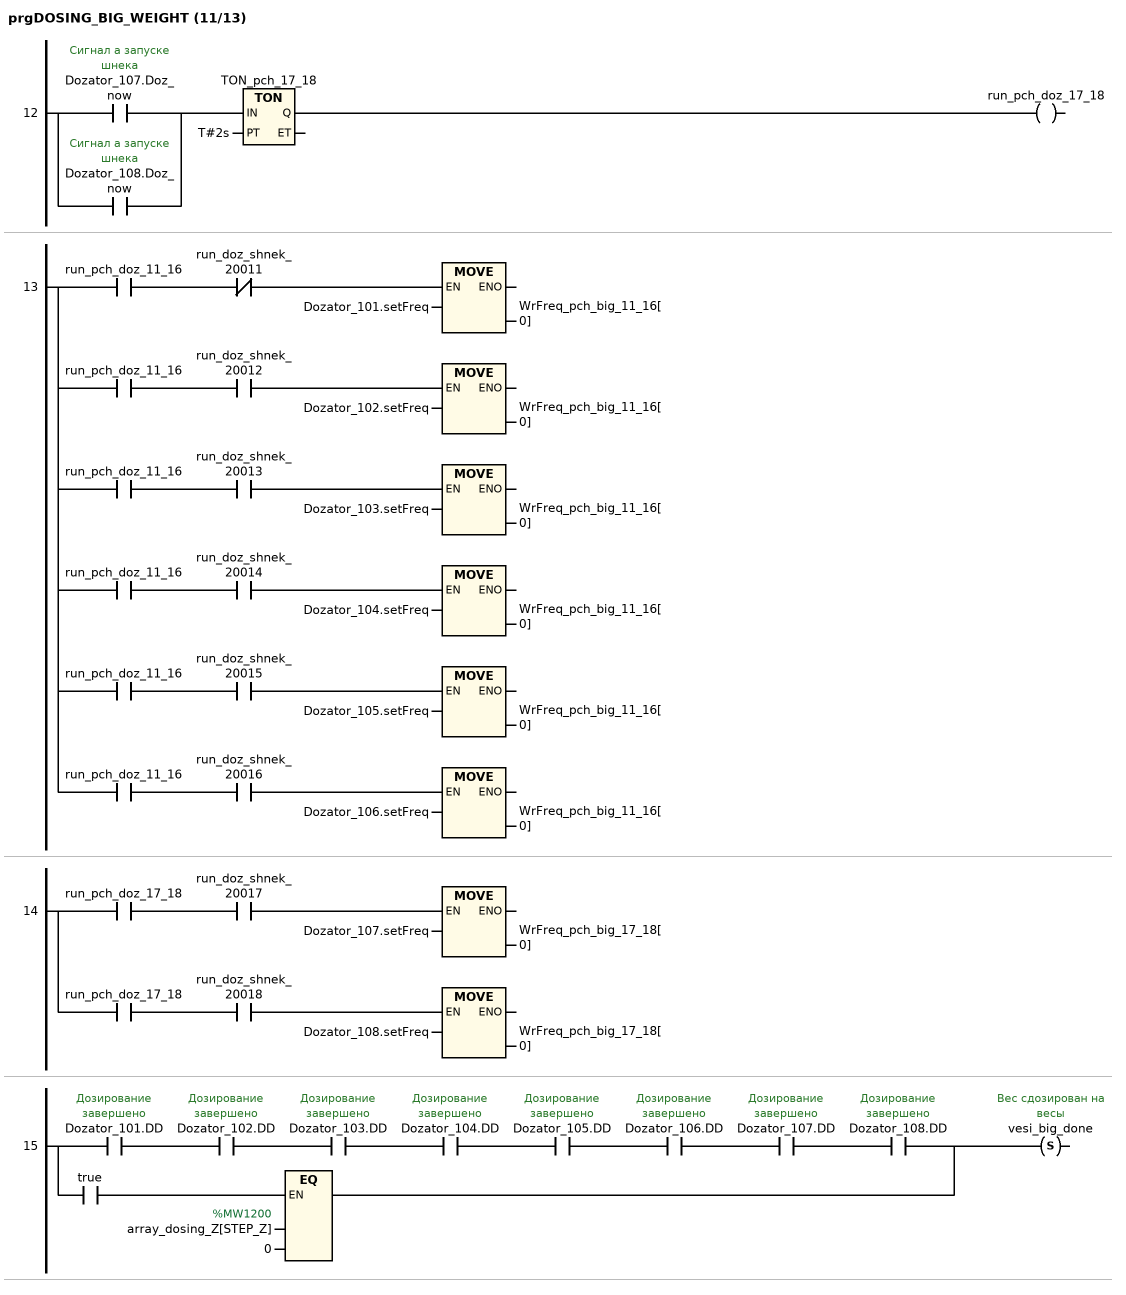
// NETWORK 12
//   Dozator_107.Doz_now: Сигнал а запуске шнека
//   Dozator_108.Doz_now: Сигнал а запуске шнека
TON_pch_17_18(IN := Dozator_107.Doz_now OR Dozator_108.Doz_now, PT := T#2s); // TON
run_pch_doz_17_18 := TON_pch_17_18.Q;

// NETWORK 13
//   Dozator_101.setFreq: Частота для частотника
//   WrFreq_pch_big_11_16[0]: PCH_BIG_11_16 : Write Multiple Registers | AT %QW17
//   Dozator_102.setFreq: Частота для частотника
//   Dozator_103.setFreq: Частота для частотника
//   Dozator_104.setFreq: Частота для частотника
//   Dozator_105.setFreq: Частота для частотника
//   Dozator_106.setFreq: Частота для частотника
_w1 := run_pch_doz_11_16 AND NOT run_doz_shnek_20011;
IF _w1 THEN WrFreq_pch_big_11_16[0] := Dozator_101.setFreq; END_IF
_w2 := run_pch_doz_11_16 AND run_doz_shnek_20012;
IF _w2 THEN WrFreq_pch_big_11_16[0] := Dozator_102.setFreq; END_IF
_w3 := run_pch_doz_11_16 AND run_doz_shnek_20013;
IF _w3 THEN WrFreq_pch_big_11_16[0] := Dozator_103.setFreq; END_IF
_w4 := run_pch_doz_11_16 AND run_doz_shnek_20014;
IF _w4 THEN WrFreq_pch_big_11_16[0] := Dozator_104.setFreq; END_IF
_w5 := run_pch_doz_11_16 AND run_doz_shnek_20015;
IF _w5 THEN WrFreq_pch_big_11_16[0] := Dozator_105.setFreq; END_IF
_w6 := run_pch_doz_11_16 AND run_doz_shnek_20016;
IF _w6 THEN WrFreq_pch_big_11_16[0] := Dozator_106.setFreq; END_IF
(* _w1 OR _w2 OR _w3 OR _w4 OR _w5 OR _w6; result not used *)

// NETWORK 14
//   Dozator_107.setFreq: Частота для частотника
//   WrFreq_pch_big_17_18[0]: PCH_BIG_17_18 : Write Multiple Registers | AT %QW18
//   Dozator_108.setFreq: Частота для частотника
_w7 := run_pch_doz_17_18 AND run_doz_shnek_20017;
IF _w7 THEN WrFreq_pch_big_17_18[0] := Dozator_107.setFreq; END_IF
_w8 := run_pch_doz_17_18 AND run_doz_shnek_20018;
IF _w8 THEN WrFreq_pch_big_17_18[0] := Dozator_108.setFreq; END_IF
(* _w7 OR _w8; result not used *)

// NETWORK 15
//   Dozator_101.DD: Дозирование завершено
//   Dozator_102.DD: Дозирование завершено
//   Dozator_103.DD: Дозирование завершено
//   Dozator_104.DD: Дозирование завершено
//   Dozator_105.DD: Дозирование завершено
//   Dozator_106.DD: Дозирование завершено
//   Dozator_107.DD: Дозирование завершено
//   Dozator_108.DD: Дозирование завершено
//   array_dosing_Z[STEP_Z]: Массив очереди дозирования больших весов (в ячейке храниться номер бункера из которого нужно дозировать) | AT %MW1200
//   vesi_big_done: Вес сдозирован на весы
vesi_big_done S= Dozator_101.DD AND Dozator_102.DD AND Dozator_103.DD AND Dozator_104.DD AND Dozator_105.DD AND Dozator_106.DD AND Dozator_107.DD AND Dozator_108.DD OR true AND array_dosing_Z[STEP_Z] = 0;

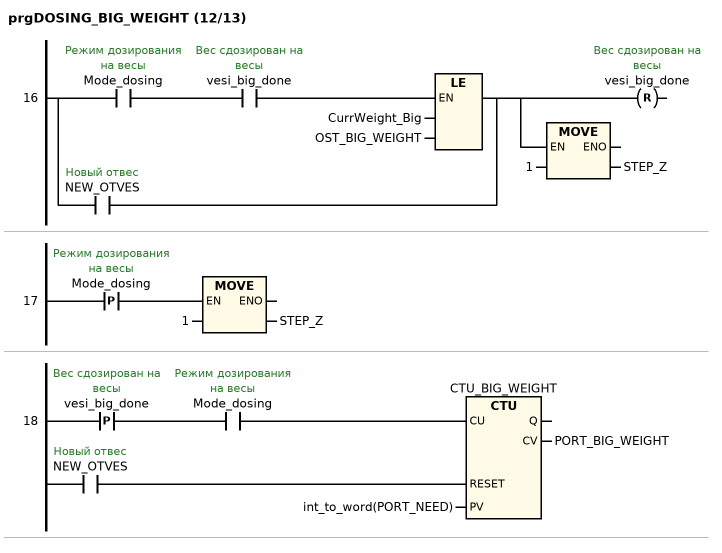
// NETWORK 16
//   Mode_dosing: Режим дозирования на весы
//   vesi_big_done: Вес сдозирован на весы
//   CurrWeight_Big: Вес на больших весах
//   OST_BIG_WEIGHT: Остаток на больших весах (вводиться со скады)
//   NEW_OTVES: Новый отвес
//   STEP_Z: Стетчик для массива очереди дозирования больших вессов
_w9 := Mode_dosing AND vesi_big_done AND CurrWeight_Big <= OST_BIG_WEIGHT OR NEW_OTVES;
vesi_big_done R= _w9;
IF _w9 THEN STEP_Z := 1; END_IF

// NETWORK 17
//   Mode_dosing: Режим дозирования на весы
//   STEP_Z: Стетчик для массива очереди дозирования больших вессов
_rt10(CLK := Mode_dosing);
IF _rt10.Q THEN STEP_Z := 1; END_IF

// NETWORK 18
//   vesi_big_done: Вес сдозирован на весы
//   Mode_dosing: Режим дозирования на весы
//   NEW_OTVES: Новый отвес
//   PORT_BIG_WEIGHT: Количество сдозированых порций на больших весах
_rt11(CLK := vesi_big_done);
CTU_BIG_WEIGHT(
    CU := _rt11.Q AND Mode_dosing,
    RESET := NEW_OTVES,
    PV := int_to_word(PORT_NEED),
    CV => PORT_BIG_WEIGHT); // CTU

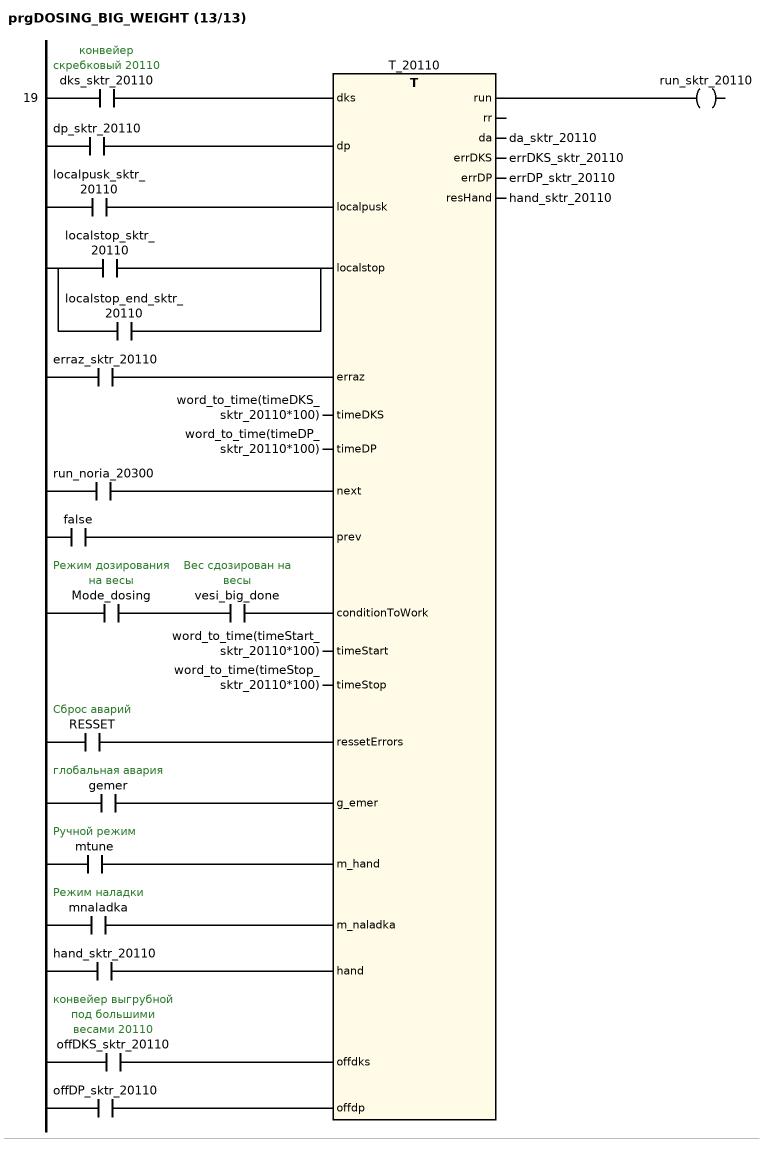
// NETWORK 19
//   dks_sktr_20110: конвейер скребковый 20110
//   Mode_dosing: Режим дозирования на весы
//   vesi_big_done: Вес сдозирован на весы
//   RESSET: Сброс аварий
//   gemer: глобальная авария
//   mtune: Ручной режим
//   mnaladka: Режим наладки
//   offDKS_sktr_20110: конвейер выгрубной под большими весами 20110
//   errDKS_sktr_20110: Конвейер выгрубной од большими весами 20110
T_20110(
    dks := dks_sktr_20110,
    dp := dp_sktr_20110,
    localpusk := localpusk_sktr_20110,
    localstop := localstop_sktr_20110 OR localstop_end_sktr_20110,
    erraz := erraz_sktr_20110,
    timeDKS := word_to_time(timeDKS_sktr_20110*100),
    timeDP := word_to_time(timeDP_sktr_20110*100),
    next := run_noria_20300,
    prev := false,
    conditionToWork := Mode_dosing AND vesi_big_done,
    timeStart := word_to_time(timeStart_sktr_20110*100),
    timeStop := word_to_time(timeStop_sktr_20110*100),
    ressetErrors := RESSET,
    g_emer := gemer,
    m_hand := mtune,
    m_naladka := mnaladka,
    hand := hand_sktr_20110,
    offdks := offDKS_sktr_20110,
    offdp := offDP_sktr_20110,
    da => da_sktr_20110,
    errDKS => errDKS_sktr_20110,
    errDP => errDP_sktr_20110,
    resHand => hand_sktr_20110); // T
run_sktr_20110 := T_20110.run;

END_PROGRAM

// PLC_241/Application/FB/SKTR/Dozator
FUNCTION_BLOCK Dozator
VAR_INPUT
	errPch: BOOL;			// Авария ПЧ
	dp: BOOL;				// Датчик подпора
	localstop: BOOL;		// Местный стоп
	conditionToWork: BOOL;	// Разрешение на запуск
	Next: BOOL;				// Сигнал, Выгребательный шнек под весами не работает (можно дозировать)
	ressetErrors: BOOL;		// Сброс аварий
	g_emer: BOOL;			// Общая глобальная авария по системе
	m_hand: BOOL;			// Ручной режим
	m_naladka: BOOL;		// Наладочный режим
	
	timeStart: TIME;		// Время через которое произойдет запуск
	timeDP: TIME;
	timeAssumptionWeight: TIME; // Время на успакоение веса
	Use: BOOL;				// Бит, нужен ли дозатор в рецепте
	Unl_done: BOOL;			// 

	Weight_Vesi: REAL;		// Текущий вес на весах
	Need_W: REAL;			// Вес который нужно сдозировать
	RA_W: REAL;				// Вес при котором переходит на точное дозирование
	Wait_W: REAL;			// Ожидаемый вес после дозирования
	Fall_weight: REAL;		// Вес падающего столба (Выбег)
	
	offdp: BOOL;			// Отключить датчик 
	hand: BOOL;				// Вкл. дазатор в ручном или наладочном режиме
	vlHIsp: WORD;			// Макс. частота дозатора
	vlLOWsp: WORD;			// Минимальная частоат дозатора
	vlPlusWeight: REAL;		// Отклонение + в кг
	vlMinusWeight: REAL;	// Отклонение - в кг
	autoKorection: BOOL;	// Автокоррекция по 5 порциям
END_VAR
VAR_OUTPUT
	run: BOOL;			// Пуск пускателя шнека
	rr: BOOL;			// готовность шнека
	da: BOOL;			// общая авария механизма
	errDP: BOOL;		// Авария датчика подпора
	Doz_now: BOOL;		// Сигнал а запуске пускателя, если есть то запускаем ПЧ
	Acc_now: BOOL;		// Переход на точное дозирование
	DD: BOOL;			// Дозирование завершено
	Corr_W : REAL;		// 
	real_W: REAL;	
	RessetPch: BOOL;	// Сброс аварии с ПЧ
	resHand: BOOL;		// Сброс бита отвечающего за запуск в ручном или наладочном режиме
	setFreq: WORD;		// Частота для частотника
	newFall: REAL;
END_VAR
VAR
	on: TON;
	off: TON;
	TP_0: TP;
	TON_1: TON;
	TOF_run: TOF;
	ghgf: BOOL;
	TON_dozdone: TON;
	TON_DP: TON;
	tmp: BOOL;
	tmpWait_w: REAL;
	TON_0: TON;
	tmpWaitDropSpeed: REAL; // Вес который нужно дозировать на снижении скорости (полный)
	oneprocWeight: REAL;	// Вес в одном проценте, который нужно дозировать на малой скорости (от полного)
	weightDOZ: REAL;		// контроля веса в снижении	(сколько сдозиравоно на снижении)
	procDOZ: REAL;			// Процент сдозированного веса	(сдозированого от полного на снижении)
	countStepDoz: INT;		// Счет порций при подсчете падающего столба (Выбега)
	
	dopusk: BOOL;			// Дозирование в допуске
	mnogo: BOOL;			// Дозирование много (пересып), нужно увеличивать падающий столб (Выбег)
	malo: BOOL;				// Дозирование мало (недосып), нужно уменьшать падающий столб (Выбег)
END_VAR
VAR // added by the converter: edge detectors and wires of the graphical bodies
    _w1, _w2, _w3, _w4, _w5, _w6, _w7, _w8 : BOOL;
    _rt1, _rt2, _rt3, _rt4 : R_TRIG;
    _ft1 : F_TRIG;
END_VAR

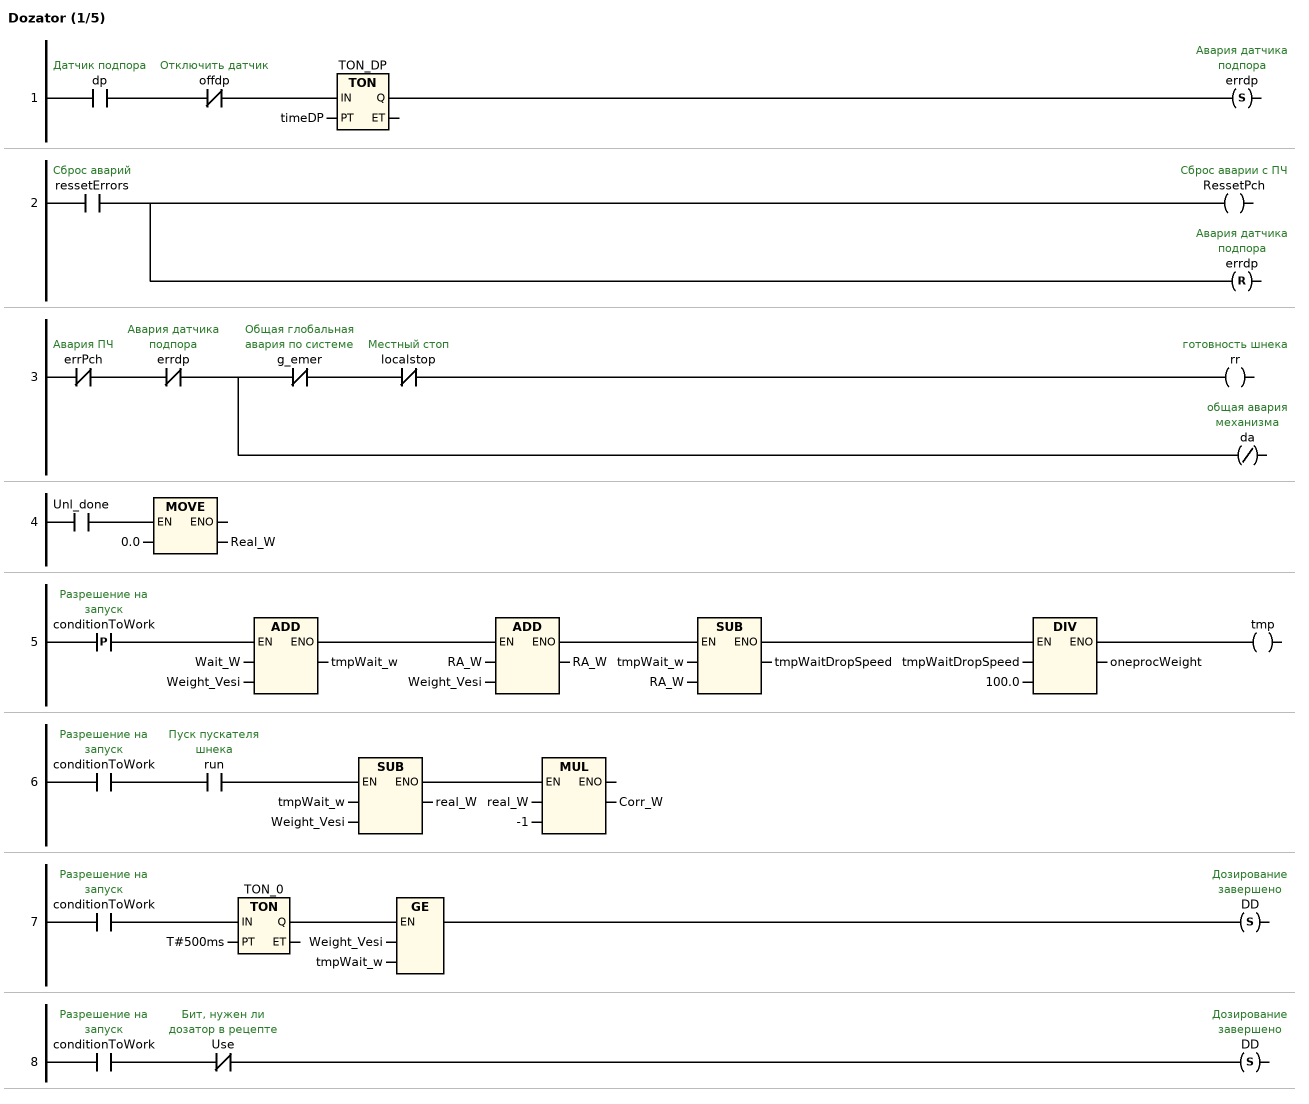
// NETWORK 1
//   dp: Датчик подпора
//   offdp: Отключить датчик
//   errdp: Авария датчика подпора
TON_DP(IN := dp AND NOT offdp, PT := timeDP); // TON
errdp S= TON_DP.Q;

// NETWORK 2
//   ressetErrors: Сброс аварий
//   RessetPch: Сброс аварии с ПЧ
//   errdp: Авария датчика подпора
RessetPch := ressetErrors;
errdp R= ressetErrors;

// NETWORK 3
//   errPch: Авария ПЧ
//   errdp: Авария датчика подпора
//   g_emer: Общая глобальная авария по системе
//   localstop: Местный стоп
//   rr: готовность шнека
//   da: общая авария механизма
_w1 := NOT errPch AND NOT errdp;
rr := _w1 AND NOT g_emer AND NOT localstop;
da := NOT _w1;

// NETWORK 4
IF Unl_done THEN Real_W := 0.0; END_IF

// NETWORK 5
//   conditionToWork: Разрешение на запуск
//   Wait_W: Ожидаемый вес после дозирования
//   Weight_Vesi: Текущий вес на весах
//   RA_W: Вес при котором переходит на точное дозирование
//   tmpWaitDropSpeed: Вес который нужно дозировать на снижении скорости (полный)
//   oneprocWeight: Вес в одном проценте, который нужно дозировать на малой скорости (от полного)
_rt1(CLK := conditionToWork);
_w2 := _rt1.Q;
IF _w2 THEN tmpWait_w := Wait_W + Weight_Vesi; END_IF
IF _w2 THEN RA_W := RA_W + Weight_Vesi; END_IF
IF _w2 THEN tmpWaitDropSpeed := tmpWait_w - RA_W; END_IF
IF _w2 THEN oneprocWeight := tmpWaitDropSpeed / 100.0; END_IF
tmp := _w2;

// NETWORK 6
//   conditionToWork: Разрешение на запуск
//   run: Пуск пускателя шнека
//   Weight_Vesi: Текущий вес на весах
_w3 := conditionToWork AND run;
IF _w3 THEN real_W := tmpWait_w - Weight_Vesi; END_IF
IF _w3 THEN Corr_W := real_W * -1; END_IF

// NETWORK 7
//   conditionToWork: Разрешение на запуск
//   Weight_Vesi: Текущий вес на весах
//   DD: Дозирование завершено
TON_0(IN := conditionToWork, PT := T#500ms); // TON
DD S= TON_0.Q AND Weight_Vesi >= tmpWait_w;

// NETWORK 8
//   conditionToWork: Разрешение на запуск
//   Use: Бит, нужен ли дозатор в рецепте
//   DD: Дозирование завершено
DD S= conditionToWork AND NOT Use;

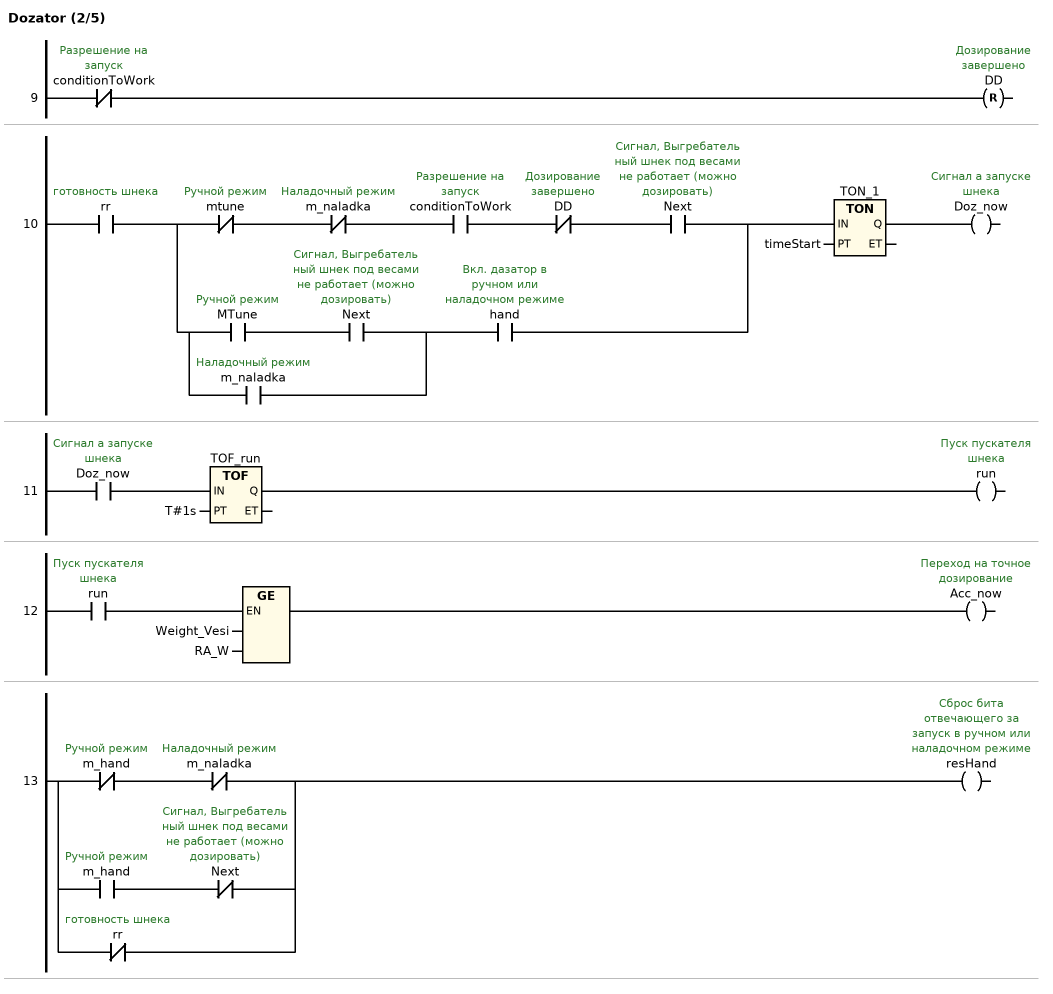
// NETWORK 9
//   conditionToWork: Разрешение на запуск
//   DD: Дозирование завершено
DD R= NOT conditionToWork;

// NETWORK 10
//   rr: готовность шнека
//   mtune: Ручной режим
//   m_naladka: Наладочный режим
//   conditionToWork: Разрешение на запуск
//   DD: Дозирование завершено
//   Next: Сигнал, Выгребательный шнек под весами не работает (можно дозировать)
//   MTune: Ручной режим
//   hand: Вкл. дазатор в ручном или наладочном режиме
//   timeStart: Время через которое произойдет запуск
//   Doz_now: Сигнал а запуске шнека
TON_1(IN := rr AND (NOT mtune AND NOT m_naladka AND conditionToWork AND NOT DD AND Next OR (MTune AND Next OR m_naladka) AND hand), PT := timeStart); // TON
Doz_now := TON_1.Q;

// NETWORK 11
//   Doz_now: Сигнал а запуске шнека
//   run: Пуск пускателя шнека
TOF_run(IN := Doz_now, PT := T#1s); // TOF
run := TOF_run.Q;

// NETWORK 12
//   run: Пуск пускателя шнека
//   Weight_Vesi: Текущий вес на весах
//   RA_W: Вес при котором переходит на точное дозирование
//   Acc_now: Переход на точное дозирование
Acc_now := run AND Weight_Vesi >= RA_W;

// NETWORK 13
//   m_hand: Ручной режим
//   m_naladka: Наладочный режим
//   Next: Сигнал, Выгребательный шнек под весами не работает (можно дозировать)
//   rr: готовность шнека
//   resHand: Сброс бита отвечающего за запуск в ручном или наладочном режиме
resHand := NOT m_hand AND NOT m_naladka OR m_hand AND NOT Next OR NOT rr;

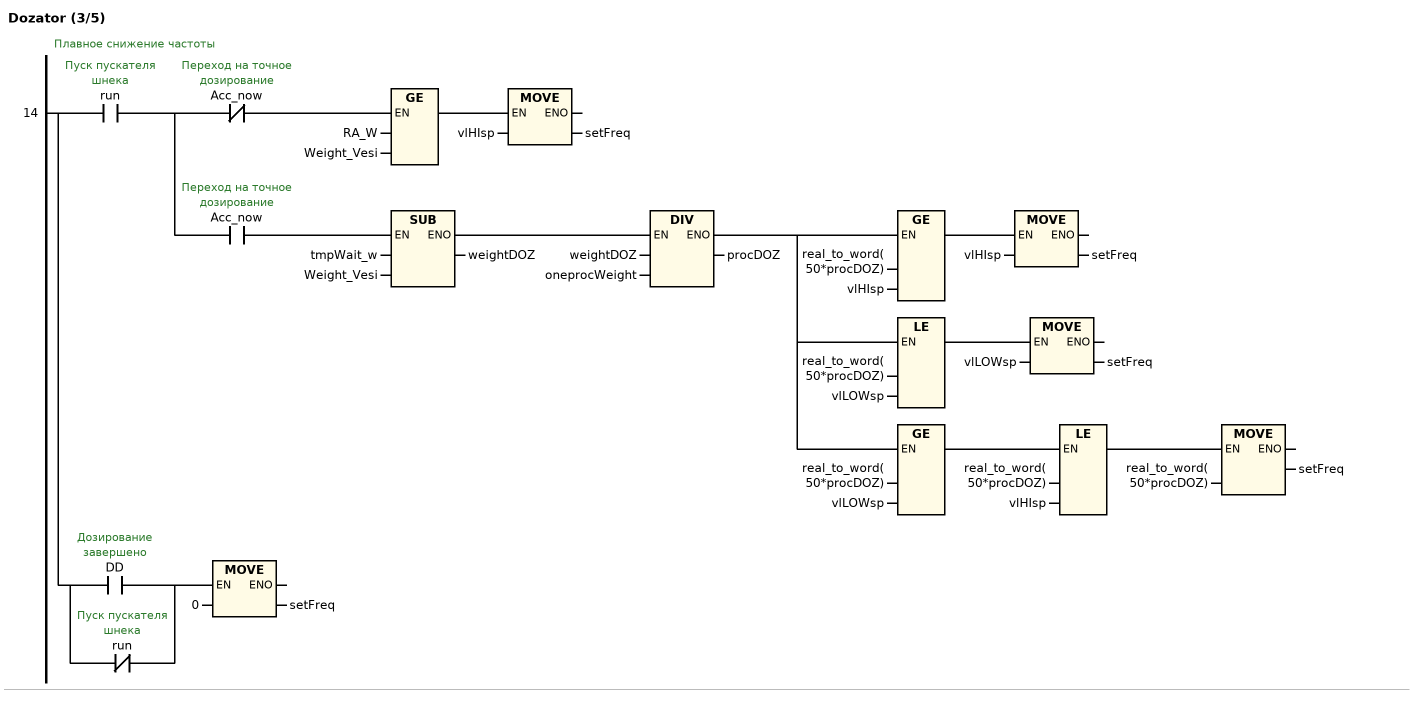
// NETWORK 14
// Плавное снижение частоты
//   run: Пуск пускателя шнека
//   Acc_now: Переход на точное дозирование
//   RA_W: Вес при котором переходит на точное дозирование
//   Weight_Vesi: Текущий вес на весах
//   vlHIsp: Макс. частота дозатора
//   setFreq: Частота для частотника
//   weightDOZ: контроля веса в снижении (сколько сдозиравоно на снижении)
//   oneprocWeight: Вес в одном проценте, который нужно дозировать на малой скорости (от полного)
//   procDOZ: Процент сдозированного веса (сдозированого от полного на снижении)
//   vlLOWsp: Минимальная частоат дозатора
//   DD: Дозирование завершено
IF run AND NOT Acc_now AND RA_W >= Weight_Vesi THEN setFreq := vlHIsp; END_IF
_w4 := run AND Acc_now;
IF _w4 THEN weightDOZ := tmpWait_w - Weight_Vesi; END_IF
IF _w4 THEN procDOZ := weightDOZ / oneprocWeight; END_IF
IF _w4 AND (real_to_word(50*procDOZ)) >= vlHIsp THEN setFreq := vlHIsp; END_IF
IF _w4 AND (real_to_word(50*procDOZ)) <= vlLOWsp THEN setFreq := vlLOWsp; END_IF
IF _w4 AND (real_to_word(50*procDOZ)) >= vlLOWsp AND (real_to_word(50*procDOZ)) <= vlHIsp THEN
    setFreq := real_to_word(50*procDOZ);
END_IF
IF DD OR NOT run THEN setFreq := 0; END_IF

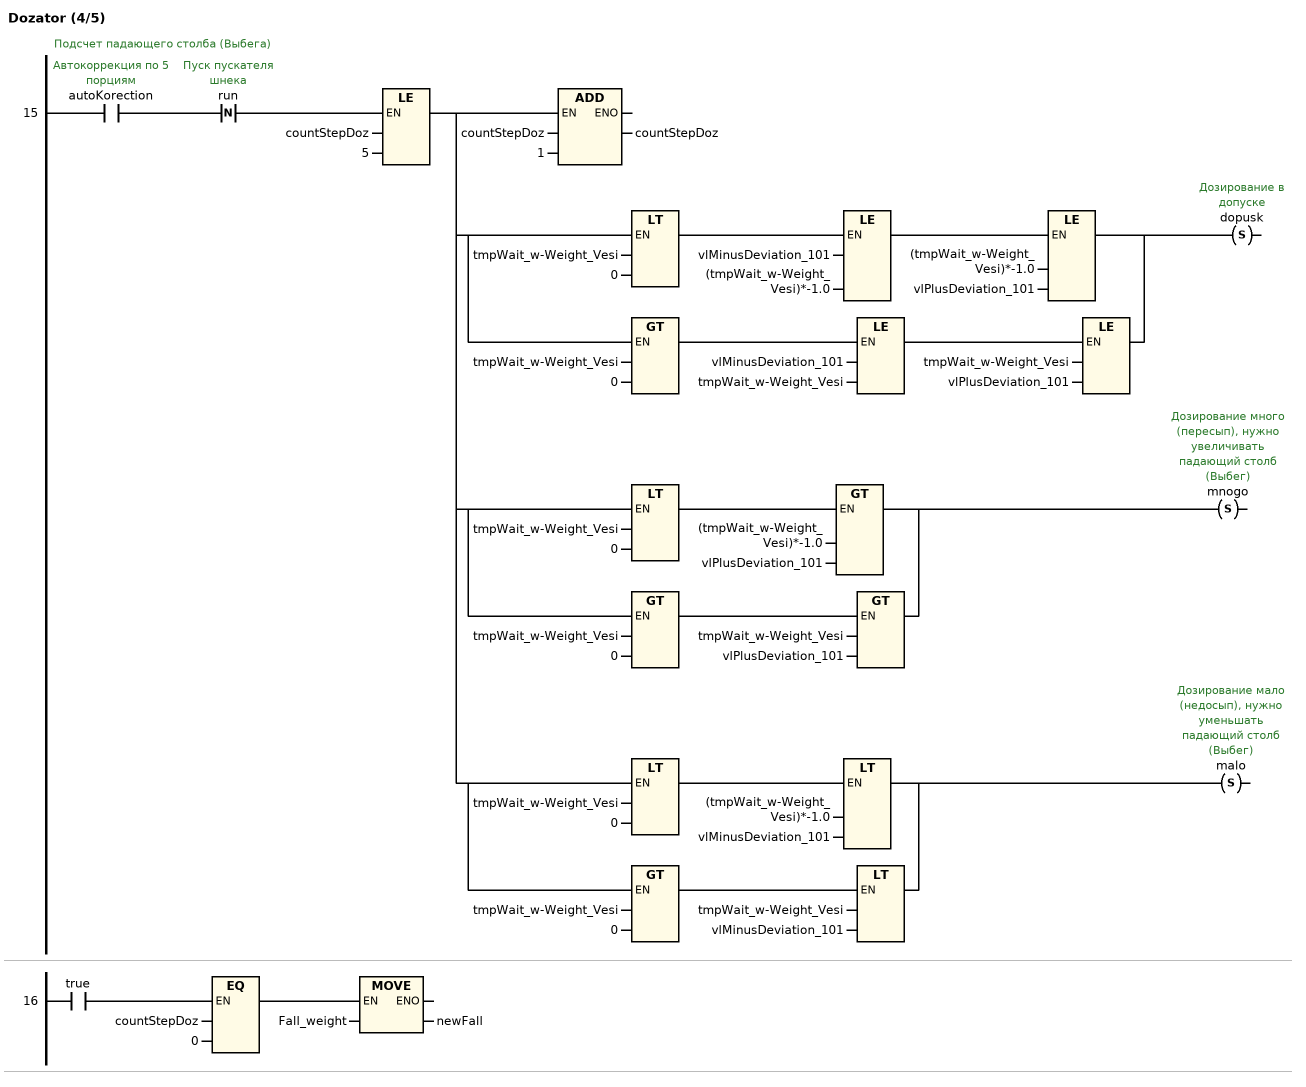
// NETWORK 15
// Подсчет падающего столба (Выбега)
//   autoKorection: Автокоррекция по 5 порциям
//   run: Пуск пускателя шнека
//   countStepDoz: Счет порций при подсчете падающего столба (Выбега)
//   vlPlusDeviation_101: ----------------------------------------------------------------------------------------------------- Значение (кг) допустимое отклонение +/- каждого компонента -----------------------------------------------------------------------------------------------------
//   dopusk: Дозирование в допуске
//   mnogo: Дозирование много (пересып), нужно увеличивать падающий столб (Выбег)
//   malo: Дозирование мало (недосып), нужно уменьшать падающий столб (Выбег)
_ft1(CLK := run);
_w5 := autoKorection AND _ft1.Q AND countStepDoz <= 5;
IF _w5 THEN countStepDoz := countStepDoz + 1; END_IF
dopusk S= _w5 AND (tmpWait_w-Weight_Vesi) < 0 AND vlMinusDeviation_101 <= ((tmpWait_w-Weight_Vesi)*-1.0) AND ((tmpWait_w-Weight_Vesi)*-1.0) <= vlPlusDeviation_101 OR _w5 AND (tmpWait_w-Weight_Vesi) > 0 AND vlMinusDeviation_101 <= (tmpWait_w-Weight_Vesi) AND (tmpWait_w-Weight_Vesi) <= vlPlusDeviation_101;
mnogo S= _w5 AND (tmpWait_w-Weight_Vesi) < 0 AND ((tmpWait_w-Weight_Vesi)*-1.0) > vlPlusDeviation_101 OR _w5 AND (tmpWait_w-Weight_Vesi) > 0 AND (tmpWait_w-Weight_Vesi) > vlPlusDeviation_101;
malo S= _w5 AND (tmpWait_w-Weight_Vesi) < 0 AND ((tmpWait_w-Weight_Vesi)*-1.0) < vlMinusDeviation_101 OR _w5 AND (tmpWait_w-Weight_Vesi) > 0 AND (tmpWait_w-Weight_Vesi) < vlMinusDeviation_101;

// NETWORK 16
//   countStepDoz: Счет порций при подсчете падающего столба (Выбега)
//   Fall_weight: Вес падающего столба (Выбег)
IF true AND countStepDoz = 0 THEN newFall := Fall_weight; END_IF

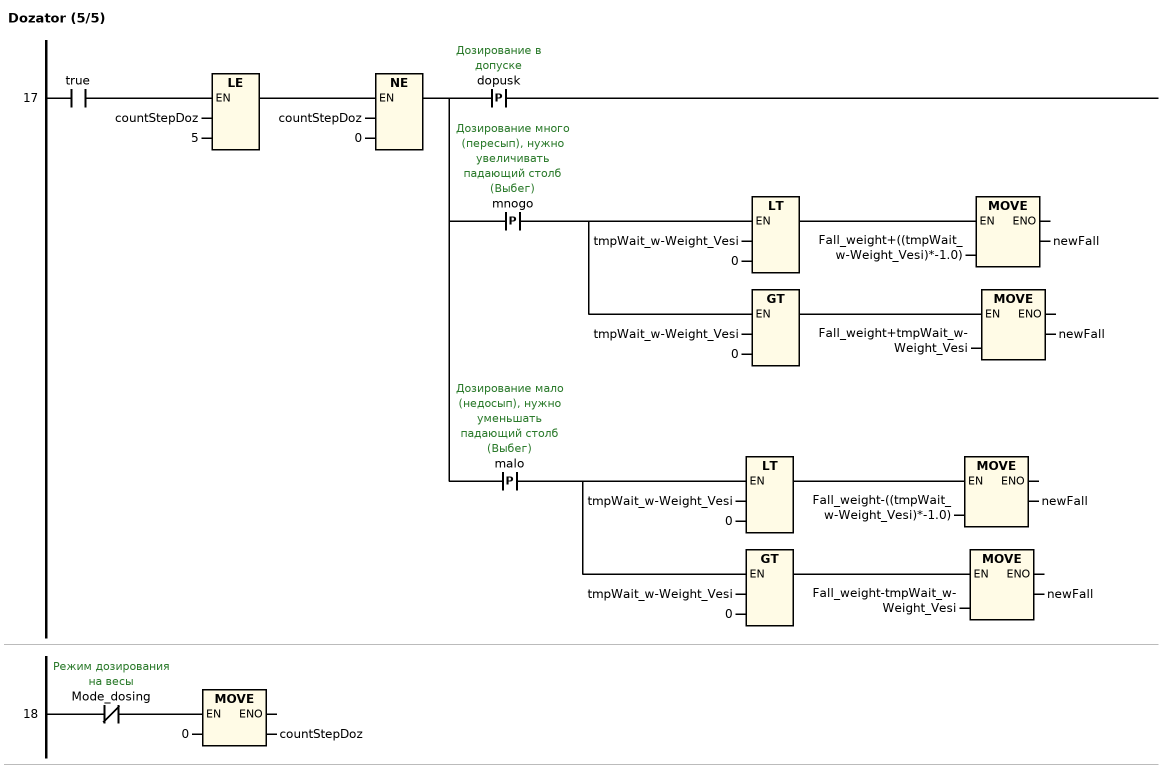
// NETWORK 17
//   countStepDoz: Счет порций при подсчете падающего столба (Выбега)
//   dopusk: Дозирование в допуске
//   mnogo: Дозирование много (пересып), нужно увеличивать падающий столб (Выбег)
//   Fall_weight+((tmpWait_w-Weight_Vesi)*-1.0): Вес падающего столба (Выбег)
//   Fall_weight+tmpWait_w-Weight_Vesi: Вес падающего столба (Выбег)
//   malo: Дозирование мало (недосып), нужно уменьшать падающий столб (Выбег)
//   Fall_weight-((tmpWait_w-Weight_Vesi)*-1.0): Вес падающего столба (Выбег)
//   Fall_weight-tmpWait_w-Weight_Vesi: Вес падающего столба (Выбег)
_w6 := true AND countStepDoz <= 5 AND countStepDoz <> 0;
_rt2(CLK := dopusk);
(* _w6 AND _rt2.Q; result not used *)
_rt3(CLK := mnogo);
_w7 := _w6 AND _rt3.Q;
IF _w7 AND (tmpWait_w-Weight_Vesi) < 0 THEN newFall := Fall_weight+((tmpWait_w-Weight_Vesi)*-1.0); END_IF
IF _w7 AND (tmpWait_w-Weight_Vesi) > 0 THEN newFall := Fall_weight+tmpWait_w-Weight_Vesi; END_IF
_rt4(CLK := malo);
_w8 := _w6 AND _rt4.Q;
IF _w8 AND (tmpWait_w-Weight_Vesi) < 0 THEN newFall := Fall_weight-((tmpWait_w-Weight_Vesi)*-1.0); END_IF
IF _w8 AND (tmpWait_w-Weight_Vesi) > 0 THEN newFall := Fall_weight-tmpWait_w-Weight_Vesi; END_IF

// NETWORK 18
//   Mode_dosing: Режим дозирования на весы
//   countStepDoz: Счет порций при подсчете падающего столба (Выбега)
IF NOT Mode_dosing THEN countStepDoz := 0; END_IF

END_FUNCTION_BLOCK

// PLC_241/Application/Recept
PROGRAM Recept
VAR
	OST: INT;
	array_port_weight: ARRAY[1..2000] OF REAL;
	newCountPort: INT;
	i: INT;
	tmpPortNeed: INT;
END_VAR


	IF Weight_PORCIA > 0 THEN
	// Подсчет целых порций
		tmpPortNeed:= Weight_PATH / Weight_PORCIA;
		ELSE
			PORT_NEED:= 0;
	END_IF
	
// Остаток 
	OST:= Weight_PATH - (tmpPortNeed * Weight_PORCIA);
	
	IF OST <= 500 AND OST < 1500 THEN
		newCountPort:= (OST + Weight_PORCIA)/2;
		FOR i:=1 TO tmpPortNeed+1 DO
			
			IF i < tmpPortNeed THEN
				array_port_weight[i]:= Weight_PORCIA;
				ELSE
					array_port_weight[i]:= newCountPort;
			END_IF
		END_FOR
		ELSE
			FOR i:= 1 TO tmpPortNeed+1 DO
				IF i<=tmpPortNeed THEN
					array_port_weight[i]:= Weight_PORCIA;
					ELSE
						array_port_weight[i]:= OST;
				END_IF
			END_FOR
	END_IF
	
	if tmpPortNeed > 0 and OST = 0 then PORT_NEED:= tmpPortNeed; end_if;
	if tmpPortNeed > 0 and OST > 0 then PORT_NEED:= tmpPortNeed+1; end_if;
	
// Вычиcляем сколько кг в одном проценте
	one_procent:= array_port_weight[PORT_BIG_WEIGHT+1]/100.0;
	
// Перещет компонентов
	K_101:= KP_101 * one_procent; 
	K_102:= KP_102 * one_procent;
	K_103:= KP_103 * one_procent;
	K_104:= KP_104 * one_procent;
	K_105:= KP_105 * one_procent;
	K_106:= KP_106 * one_procent;
	K_107:= KP_107 * one_procent;
	K_108:= KP_108 * one_procent;
		
	IF K_101 > 0 THEN Use_101:= TRUE; ELSE Use_101:= FALSE; END_IF;
	IF K_102 > 0 THEN Use_102:= TRUE; ELSE Use_102:= FALSE; END_IF;
	IF K_103 > 0 THEN Use_103:= TRUE; ELSE Use_103:= FALSE; END_IF;
	IF K_104 > 0 THEN Use_104:= TRUE; ELSE Use_104:= FALSE; END_IF;
	IF K_105 > 0 THEN Use_105:= TRUE; ELSE Use_105:= FALSE; END_IF;
	IF K_106 > 0 THEN Use_106:= TRUE; ELSE Use_106:= FALSE; END_IF;
	IF K_107 > 0 THEN Use_107:= TRUE; ELSE Use_107:= FALSE; END_IF;
	IF K_108 > 0 THEN Use_108:= TRUE; ELSE Use_108:= FALSE; END_IF;
		
// Расчет процентного отклонения компонентов
	IF K_101 <> 0 THEN vlPlusDeviation_101:= K_101/100.0 * (INT_TO_REAL(ivlPlusDeviation_101)/10.0); ELSE vlPlusDeviation_101:= 0; END_IF;
	IF K_102 <> 0 THEN vlPlusDeviation_102:= K_102/100.0 * (INT_TO_REAL(ivlPlusDeviation_102)/10.0); ELSE vlPlusDeviation_102:= 0; END_IF;
	IF K_103 <> 0 THEN vlPlusDeviation_103:= K_103/100.0 * (INT_TO_REAL(ivlPlusDeviation_103)/10.0); ELSE vlPlusDeviation_103:= 0; END_IF;
	IF K_104 <> 0 THEN vlPlusDeviation_104:= K_104/100.0 * (INT_TO_REAL(ivlPlusDeviation_104)/10.0); ELSE vlPlusDeviation_104:= 0; END_IF;
	IF K_105 <> 0 THEN vlPlusDeviation_105:= K_105/100.0 * (INT_TO_REAL(ivlPlusDeviation_105)/10.0); ELSE vlPlusDeviation_105:= 0; END_IF;
	IF K_106 <> 0 THEN vlPlusDeviation_106:= K_106/100.0 * (INT_TO_REAL(ivlPlusDeviation_106)/10.0); ELSE vlPlusDeviation_106:= 0; END_IF;
	IF K_107 <> 0 THEN vlPlusDeviation_107:= K_107/100.0 * (INT_TO_REAL(ivlPlusDeviation_107)/10.0); ELSE vlPlusDeviation_107:= 0; END_IF;
	IF K_108 <> 0 THEN vlPlusDeviation_108:= K_108/100.0 * (INT_TO_REAL(ivlPlusDeviation_108)/10.0); ELSE vlPlusDeviation_108:= 0; END_IF;
		
	IF K_101 <> 0 THEN vlMinusDeviation_101:= K_101/100.0 * (INT_TO_REAL(ivlMinusDeviation_101)/10.0); ELSE vlMinusDeviation_101:= 0; END_IF;
	IF K_102 <> 0 THEN vlMinusDeviation_102:= K_102/100.0 * (INT_TO_REAL(ivlMinusDeviation_102)/10.0); ELSE vlMinusDeviation_102:= 0; END_IF;
	IF K_103 <> 0 THEN vlMinusDeviation_103:= K_103/100.0 * (INT_TO_REAL(ivlMinusDeviation_103)/10.0); ELSE vlMinusDeviation_103:= 0; END_IF;
	IF K_104 <> 0 THEN vlMinusDeviation_104:= K_104/100.0 * (INT_TO_REAL(ivlMinusDeviation_104)/10.0); ELSE vlMinusDeviation_104:= 0; END_IF;
	IF K_105 <> 0 THEN vlMinusDeviation_105:= K_105/100.0 * (INT_TO_REAL(ivlMinusDeviation_105)/10.0); ELSE vlMinusDeviation_105:= 0; END_IF;
	IF K_106 <> 0 THEN vlMinusDeviation_106:= K_106/100.0 * (INT_TO_REAL(ivlMinusDeviation_106)/10.0); ELSE vlMinusDeviation_106:= 0; END_IF;
	IF K_107 <> 0 THEN vlMinusDeviation_107:= K_107/100.0 * (INT_TO_REAL(ivlMinusDeviation_107)/10.0); ELSE vlMinusDeviation_107:= 0; END_IF;
	IF K_108 <> 0 THEN vlMinusDeviation_108:= K_108/100.0 * (INT_TO_REAL(ivlMinusDeviation_108)/10.0); ELSE vlMinusDeviation_108:= 0; END_IF;

END_PROGRAM

// PLC_241/Application/POU/MotoHours
PROGRAM MotoHours
VAR
	imp: Standard.R_TRIG;
END_VAR

imp(CLK:= PLC_R.i_x1sClk);

	MH_sktr_10110:= funStepMH(imp:= imp.Q, run:= run_sktr_10110, MH:= MH_sktr_10110);
	MH_AC_1_1:= funStepMH(imp:= imp.Q, run:= run_fans_AC_hole, MH:= MH_AC_1_1);
	MH_AC_1_2:= funStepMH(imp:= imp.Q, run:= run_fans_AC_hole, MH:= MH_AC_1_2);
	MH_Noria_10200:= funStepMH(imp:= imp.Q, run:= run_noria_10200, MH:= MH_Noria_10200);
	MH_LF_Noria_10200:= funStepMH(imp:= imp.Q, run:= run_AC_10201, MH:= MH_LF_Noria_10200);
	MH_Scalp:= funStepMH(imp:= imp.Q, run:= run_scalp AND run_pch_scalp, MH:= MH_Scalp);
	MH_Noria_10400:= funStepMH(imp:= imp.Q, run:= run_noria_10400, MH:= MH_Noria_10400);
	MH_LF_Noria_10400:= funStepMH(imp:= imp.Q, run:= run_AC_10401, MH:= MH_LF_Noria_10400);
	MH_sktr_10500:= funStepMH(imp:= imp.Q, run:= run_sktr_10500, MH:= MH_sktr_10500);
	MH_LF_sktr_10500:= funStepMH(imp:= imp.Q, run:= run_AC_10501, MH:= MH_LF_sktr_10500);
	MH_SH_10610:= funStepMH(imp:= imp.Q, run:= run_open_sh_10610 OR run_close_sh_10610, MH:= MH_SH_10610);
	MH_SH_10620:= funStepMH(imp:= imp.Q, run:= run_open_sh_10620 OR run_close_sh_10620, MH:= MH_SH_10620);
	MH_SH_10630:= funStepMH(imp:= imp.Q, run:= run_open_sh_10630 OR run_close_sh_10630, MH:= MH_SH_10630);
	MH_SH_10640:= funStepMH(imp:= imp.Q, run:= run_open_sh_10640 OR run_close_sh_10640, MH:= MH_SH_10640);
	MH_doz_shnek_20011:= funStepMH(imp:= imp.Q, run:= run_pch_doz_11_16 AND run_doz_shnek_20011, MH:= MH_doz_shnek_20011);
	MH_doz_shnek_20012:= funStepMH(imp:= imp.Q, run:= run_pch_doz_11_16 AND run_doz_shnek_20012, MH:= MH_doz_shnek_20012);
	MH_doz_shnek_20013:= funStepMH(imp:= imp.Q, run:= run_pch_doz_11_16 AND run_doz_shnek_20013, MH:= MH_doz_shnek_20013);
	MH_doz_shnek_20014:= funStepMH(imp:= imp.Q, run:= run_pch_doz_11_16 AND run_doz_shnek_20014, MH:= MH_doz_shnek_20014);
	MH_doz_shnek_20015:= funStepMH(imp:= imp.Q, run:= run_pch_doz_11_16 AND run_doz_shnek_20015, MH:= MH_doz_shnek_20015);
	MH_doz_shnek_20016:= funStepMH(imp:= imp.Q, run:= run_pch_doz_11_16 AND run_doz_shnek_20016, MH:= MH_doz_shnek_20016);
	MH_doz_shnek_20017:= funStepMH(imp:= imp.Q, run:= run_pch_doz_11_16 AND run_doz_shnek_20017, MH:= MH_doz_shnek_20017);
	MH_doz_shnek_20018:= funStepMH(imp:= imp.Q, run:= run_pch_doz_11_16 AND run_doz_shnek_20018, MH:= MH_doz_shnek_20018);
	MH_sktr_20110:= funStepMH(imp:= imp.Q, run:= run_sktr_20110, MH:= MH_sktr_20110);
	MH_Noria_20300:= funStepMH(imp:= imp.Q, run:= run_noria_20300, MH:= MH_Noria_20300);
	MH_LF_Noria_20301:= funStepMH(imp:= imp.Q, run:= run_AC_20301, MH:= MH_LF_Noria_20301);
	MH_SH_30110:= funStepMH(imp:= imp.Q, run:= run_open_sh_30110 OR run_close_sh_30110, MH:= MH_SH_30110);
	MH_doz_pit_drob:= funStepMH(imp:= imp.Q, run:= run_pch_30200 AND run_pit_30200, MH:= MH_doz_pit_drob);
	MH_drob:= funStepMH(imp:= imp.Q, run:= run_drob, MH:= MH_drob);
	MH_shnek_30330:= funStepMH(imp:= imp.Q, run:= run_shnek_30330, MH:= MH_shnek_30330);
	MH_shluz_30340:= funStepMH(imp:= imp.Q, run:= run_shluz_30340, MH:= MH_shluz_30340);
	MH_asp_drob_30310:= funStepMH(imp:= imp.Q, run:= run_AC_30310, MH:= MH_asp_drob_30310);
	MH_sktr_30400:= funStepMH(imp:= imp.Q, run:= run_sktr_30400, MH:= MH_sktr_30400);
	MH_Noria_21200:= funStepMH(imp:= imp.Q, run:= run_noria_21200, MH:= MH_Noria_21200);
	MH_shnek_21300:= funStepMH(imp:= imp.Q, run:= run_shnek_21300, MH:= MH_shnek_21300);
	MH_SH_21310:= funStepMH(imp:= imp.Q, run:= run_open_sh_21310 OR run_close_sh_21310, MH:= MH_SH_21310);
	MH_SH_21320:= funStepMH(imp:= imp.Q, run:= run_open_sh_21320 OR run_close_sh_21320, MH:= MH_SH_21320);
	MH_SH_21330:= funStepMH(imp:= imp.Q, run:= run_open_sh_21330 OR run_close_sh_21330, MH:= MH_SH_21330);
	MH_doz_shnek_21410:= funStepMH(imp:= imp.Q, run:= run_pch_doz_shnek_5_9 AND run_doz_shnek_21405, MH:= MH_doz_shnek_21410);
	MH_doz_shnek_21411:= funStepMH(imp:= imp.Q, run:= run_pch_doz_shnek_5_9 AND run_doz_shnek_21406, MH:= MH_doz_shnek_21411);
	MH_doz_shnek_21412:= funStepMH(imp:= imp.Q, run:= run_pch_doz_shnek_5_9 AND run_doz_shnek_21407, MH:= MH_doz_shnek_21412);
	MH_doz_shnek_21413:= funStepMH(imp:= imp.Q, run:= run_pch_doz_shnek_5_9 AND run_doz_shnek_21408, MH:= MH_doz_shnek_21413);
	MH_doz_shnek_21414:= funStepMH(imp:= imp.Q, run:= run_pch_doz_shnek_5_9 AND run_doz_shnek_21409, MH:= MH_doz_shnek_21414);
	MH_doz_shnek_21510:= funStepMH(imp:= imp.Q, run:= run_pch_doz_shnek_51_54 AND run_doz_shnek_21510, MH:= MH_doz_shnek_21510);
	MH_doz_shnek_21520:= funStepMH(imp:= imp.Q, run:= run_pch_doz_shnek_51_54 AND run_doz_shnek_21520, MH:= MH_doz_shnek_21520);
	MH_doz_shnek_21530:= funStepMH(imp:= imp.Q, run:= run_pch_doz_shnek_51_54 AND run_doz_shnek_21530, MH:= MH_doz_shnek_21530);
	MH_doz_shnek_21540:= funStepMH(imp:= imp.Q, run:= run_pch_doz_shnek_51_54 AND run_doz_shnek_21540, MH:= MH_doz_shnek_21540);
	MH_shnek_21600:= funStepMH(imp:= imp.Q, run:= run_shnek_21600, MH:= MH_shnek_21600);
	MH_Noria_30500:= funStepMH(imp:= imp.Q, run:= run_noria_30500, MH:= MH_Noria_30500);
	MH_Smes:= funStepMH(imp:= imp.Q, run:= run_smes, MH:= MH_Smes);
	MH_shnek_30640:= funStepMH(imp:= imp.Q, run:= run_shnek_30640, MH:= MH_shnek_30640);
	MH_Noria_30700:= funStepMH(imp:= imp.Q, run:= run_noria_30700, MH:= MH_Noria_30700);
	MH_LF_Noria_30700:= funStepMH(imp:= imp.Q, run:= run_AC_30701, MH:= MH_LF_Noria_30700);
	MH_sktr_30900:= funStepMH(imp:= imp.Q, run:= run_sktr_30900, MH:= MH_sktr_30900);
	MH_LF_sktr_30900:= funStepMH(imp:= imp.Q, run:= run_AC_30901, MH:= MH_LF_sktr_30900);
	MH_SH_30910:= funStepMH(imp:= imp.Q, run:= run_open_sh_30910 OR run_close_sh_30910, MH:= MH_SH_30910);
	MH_SH_30920:= funStepMH(imp:= imp.Q, run:= run_open_sh_30920 OR run_close_sh_30920, MH:= MH_SH_30920);
	MH_SH_30930:= funStepMH(imp:= imp.Q, run:= run_open_sh_30930 OR run_close_sh_30930, MH:= MH_SH_30930);
	MH_SH_30940:= funStepMH(imp:= imp.Q, run:= run_open_sh_30940 OR run_close_sh_30940, MH:= MH_SH_30940);
	MH_sktr_30800:= funStepMH(imp:= imp.Q, run:= run_sktr_30800, MH:= MH_sktr_30800);
	MH_SH_30810:= funStepMH(imp:= imp.Q, run:= run_open_sh_30810 OR run_close_sh_30810, MH:= MH_SH_30810);
	MH_SH_30820:= funStepMH(imp:= imp.Q, run:= run_open_sh_30820 OR run_close_sh_30820, MH:= MH_SH_30820);
	MH_KP_10210:= funStepMH(imp:= imp.Q, run:= run_tflap_noria_10210 OR run_tflap_scalp_10210, MH:= MH_KP_10210);
	MH_KP_10710:= funStepMH(imp:= imp.Q, run:= run_tflap_bunk_20001_10710 OR run_tflap_bunk_20002_10710, MH:= MH_KP_10710);
	MH_KP_10720:= funStepMH(imp:= imp.Q, run:= run_tflap_bunk_20003_10720 OR run_tflap_bunk_20004_10720, MH:= MH_KP_10720);
	MH_KP_10730:= funStepMH(imp:= imp.Q, run:= run_tflap_bunk_20005_10730 OR run_tflap_bunk_20006_10730, MH:= MH_KP_10730);
	MH_KP_10740:= funStepMH(imp:= imp.Q, run:= run_tflap_bunk_20007_10740 OR run_tflap_bunk_20008_10740, MH:= MH_KP_10740);

END_PROGRAM

// PLC_241/Application/funStepMH
FUNCTION funStepMH : DINT
VAR_INPUT
imp: BOOL;
run: BOOL;
MH: DINT;
END_VAR
VAR
	MM: DINT;
	result: DINT;
END_VAR

IF imp AND run THEN
	MM:= MM+1;
	IF MM >= 3600 THEN
		MH:= MH + 1;
		MM:= 0;
	END_IF
END_IF
result:= MH;
funStepMH:= result;

END_FUNCTION

// PLC_241/Application/vsState
PROGRAM vsState
VAR
	vsState_LF_ON AT %MW5000: WORD;
	vsState_LF_DA AT %MW5001: WORD;
	
	vsState_DVU_101_108 AT %MW5002: WORD;
	vsState_DNU_101_108 AT %MW5003: WORD;
	
	vsState_Noria_ON AT %MW5004: WORD;
	vsState_Noria_DA AT %MW5005: WORD;
	
	vsState_SKTR_ON AT %MW5006: WORD;
	vsState_SKTR_DA AT %MW5007: WORD;
	
	vsState_Line_load_K AT %MW5008: WORD;
	vsState_Line_load_K1 AT %MW5009: WORD;
	vsState_Line_load_K2 AT %MW5010: WORD;
	
	vsState_Z_opened AT %MW5012: WORD;
	vsState_Z_closed AT %MW5013: WORD;
	vsState_Z_per AT %MW5014: WORD;
	vsState_Z_DA AT %MW5015: WORD;
		
	vsState_KP_pol_1 AT %MW5016: WORD;
	vsState_KP_pol_2 AT %MW5017: WORD;
	vsState_KP_per AT %MW5018: WORD;
	vsState_KP_DA AT %MW5019: WORD;
	vsState_emer AT %MW5020: WORD;
	vsState_emer1 AT %MW5021: WORD;
	vsState_emer2 AT %MW5022: WORD;
END_VAR

// Работа системы локальных фильтров
	vsState_LF_ON.0:= run_fans_AC_hole;
	vsState_LF_ON.1:= run_fans_AC_hole;
	vsState_LF_ON.2:= run_AC_10201;
	vsState_LF_ON.3:= run_AC_10401;
	vsState_LF_ON.4:= run_AC_10501;
	vsState_LF_ON.5:= run_AC_30701;
	vsState_LF_ON.6:= run_AC_30901;
	vsState_LF_ON.7:= run_AC_20301;
	vsState_LF_ON.8:= FALSE;
	vsState_LF_ON.9:= FALSE;
	vsState_LF_ON.10:= FALSE;
	vsState_LF_ON.11:= FALSE;
	vsState_LF_ON.12:= FALSE;
	vsState_LF_ON.13:= FALSE;
	vsState_LF_ON.14:= FALSE;
	vsState_LF_ON.15:= FALSE;
	
// Аварии системы локальных фильтров
	vsState_LF_DA.0:= da_fans_AC_hole;
	vsState_LF_DA.1:= da_fans_AC_hole;
	vsState_LF_DA.2:= da_AC_10201;
	vsState_LF_DA.3:= da_AC_10401;
	vsState_LF_DA.4:= da_AC_10501;
	vsState_LF_DA.5:= da_AC_30701;
	vsState_LF_DA.6:= da_AC_30901;
	vsState_LF_DA.7:= da_AC_20301;
	vsState_LF_DA.8:= FALSE;
	vsState_LF_DA.9:= FALSE;
	vsState_LF_DA.10:= FALSE;
	vsState_LF_DA.11:= FALSE;
	vsState_LF_DA.12:= FALSE;
	vsState_LF_DA.13:= FALSE;
	vsState_LF_DA.14:= FALSE;
	vsState_LF_DA.15:= FALSE;
	
// Датчики верхнего уровня бункеров 101-108
	vsState_DVU_101_108.0:= dvy_bunk_101;
	vsState_DVU_101_108.1:= dvy_bunk_102;
	vsState_DVU_101_108.2:= dvy_bunk_103;
	vsState_DVU_101_108.3:= dvy_bunk_104;
	vsState_DVU_101_108.4:= dvy_bunk_105;
	vsState_DVU_101_108.5:= dvy_bunk_106;
	vsState_DVU_101_108.6:= dvy_bunk_107;
	vsState_DVU_101_108.7:= dvy_bunk_108;
	vsState_DVU_101_108.8:= dvy_bunk_201;
	vsState_DVU_101_108.9:= dvy_bunk_202;
	vsState_DVU_101_108.10:= dvy_bunk_203;
	vsState_DVU_101_108.11:= dvy_bunk_204;
	vsState_DVU_101_108.12:= FALSE;
	vsState_DVU_101_108.13:= FALSE;
	vsState_DVU_101_108.14:= FALSE;
	vsState_DVU_101_108.15:= FALSE;

// Датчики нижнего уровня бункеров 101-108
	vsState_DNU_101_108.0:= dny_bunk_101;
	vsState_DNU_101_108.1:= dny_bunk_102;
	vsState_DNU_101_108.2:= dny_bunk_103;
	vsState_DNU_101_108.3:= dny_bunk_104;
	vsState_DNU_101_108.4:= dny_bunk_105;
	vsState_DNU_101_108.5:= dny_bunk_106;
	vsState_DNU_101_108.6:= dny_bunk_107;
	vsState_DNU_101_108.7:= dny_bunk_108;
	vsState_DNU_101_108.8:= dny_bunk_201;
	vsState_DNU_101_108.9:= dny_bunk_202;
	vsState_DNU_101_108.10:= dny_bunk_203;
	vsState_DNU_101_108.11:= dny_bunk_204;
	vsState_DNU_101_108.12:= dny_hole;
	vsState_DNU_101_108.13:= FALSE;
	vsState_DNU_101_108.14:= FALSE;
	vsState_DNU_101_108.15:= FALSE;
	
// Нории
	// работа
	vsState_Noria_ON.0:= run_noria_10200;
	vsState_Noria_ON.1:= run_noria_10400;
	vsState_Noria_ON.2:= run_noria_21200;
	vsState_Noria_ON.3:= run_noria_30700;
	vsState_Noria_ON.4:= run_noria_20300;
	vsState_Noria_ON.5:= run_noria_30500;
	vsState_Noria_ON.6:= FALSE;
	vsState_Noria_ON.7:= FALSE;
	vsState_Noria_ON.8:= FALSE;
	vsState_Noria_ON.9:= FALSE;
	vsState_Noria_ON.10:= FALSE;
	vsState_Noria_ON.11:= FALSE;
	vsState_Noria_ON.12:= FALSE;
	vsState_Noria_ON.13:= FALSE;
	vsState_Noria_ON.14:= FALSE;
	vsState_Noria_ON.15:= FALSE;
	
	// Авария
	vsState_Noria_DA.0:= da_noria_10200;
	vsState_Noria_DA.1:= da_noria_10400;
	vsState_Noria_DA.2:= da_noria_21200;
	vsState_Noria_DA.3:= da_noria_30700;
	vsState_Noria_DA.4:= da_noria_20300;
	vsState_Noria_DA.5:= da_noria_30500;
	vsState_Noria_DA.6:= FALSE;
	vsState_Noria_DA.7:= FALSE;
	vsState_Noria_DA.8:= FALSE;
	vsState_Noria_DA.9:= FALSE;
	vsState_Noria_DA.10:= FALSE;
	vsState_Noria_DA.11:= FALSE;
	vsState_Noria_DA.12:= FALSE;
	vsState_Noria_DA.13:= FALSE;
	vsState_Noria_DA.14:= FALSE;
	vsState_Noria_DA.15:= FALSE;
	
// Конвейеры скребковые
	// работа
	vsState_SKTR_ON.0:= run_sktr_10110;
	vsState_SKTR_ON.1:= run_sktr_10500;
	vsState_SKTR_ON.2:= run_shnek_21300;
	vsState_SKTR_ON.3:= run_sktr_30900;
	vsState_SKTR_ON.4:= run_sktr_30800;
	vsState_SKTR_ON.5:= run_sktr_20110;
	vsState_SKTR_ON.6:= run_sktr_30400;
	vsState_SKTR_ON.7:= run_pch_sktr_30330;
	vsState_SKTR_ON.8:= run_shnek_30640;
	vsState_SKTR_ON.9:= run_shnek_21600;
	vsState_SKTR_ON.10:= FALSE;
	vsState_SKTR_ON.11:= FALSE;
	vsState_SKTR_ON.12:= FALSE;
	vsState_SKTR_ON.13:= FALSE;
	vsState_SKTR_ON.14:= FALSE;
	vsState_SKTR_ON.15:= FALSE;
	
	// авария
	vsState_SKTR_DA.0:= da_sktr_10110;
	vsState_SKTR_DA.1:= da_sktr_10500;
	vsState_SKTR_DA.2:= da_shnek_21300;
	vsState_SKTR_DA.3:= da_sktr_30900;
	vsState_SKTR_DA.4:= da_sktr_30800;
	vsState_SKTR_DA.5:= da_sktr_20110;
	vsState_SKTR_DA.6:= da_sktr_30400;
	vsState_SKTR_DA.7:= da_sktr_30330;
	vsState_SKTR_DA.8:= da_shnek_30640;
	vsState_SKTR_DA.9:= da_shnek_21600;
	vsState_SKTR_DA.10:= FALSE;
	vsState_SKTR_DA.11:= FALSE;
	vsState_SKTR_DA.12:= FALSE;
	vsState_SKTR_DA.13:= FALSE;
	vsState_SKTR_DA.14:= FALSE;
	vsState_SKTR_DA.15:= FALSE;
	
// 2-х ходовый клапана
	// pol_1
	vsState_KP_pol_1.0:= stPoz_scalp_10210;
	vsState_KP_pol_1.1:= stPoz_bunk1_10710;
	vsState_KP_pol_1.2:= stPoz_bunk3_10720;
	vsState_KP_pol_1.3:= stPoz_bunk5_10730;
	vsState_KP_pol_1.4:= stPoz_bunk7_10740;
	vsState_KP_pol_1.5:= FALSE;
	vsState_KP_pol_1.6:= FALSE;
	vsState_KP_pol_1.7:= FALSE;
	vsState_KP_pol_1.8:= FALSE;
	vsState_KP_pol_1.9:= FALSE;
	vsState_KP_pol_1.10:= FALSE;
	vsState_KP_pol_1.11:= FALSE;
	vsState_KP_pol_1.12:= FALSE;
	vsState_KP_pol_1.13:= FALSE;
	vsState_KP_pol_1.14:= FALSE;
	vsState_KP_pol_1.15:= FALSE;
	
	// pol_2
	vsState_KP_pol_2.0:= stPoz_noria_10210;
	vsState_KP_pol_2.1:= stPoz_bunk2_10710;
	vsState_KP_pol_2.2:= stPoz_bunk4_10720;
	vsState_KP_pol_2.3:= stPoz_bunk6_10730;
	vsState_KP_pol_2.4:= stPoz_bunk8_10740;
	vsState_KP_pol_2.5:= FALSE;
	vsState_KP_pol_2.6:= FALSE;
	vsState_KP_pol_2.7:= FALSE;
	vsState_KP_pol_2.8:= FALSE;
	vsState_KP_pol_2.9:= FALSE;
	vsState_KP_pol_2.10:= FALSE;
	vsState_KP_pol_2.11:= FALSE;
	vsState_KP_pol_2.12:= FALSE;
	vsState_KP_pol_2.13:= FALSE;
	vsState_KP_pol_2.14:= FALSE;
	vsState_KP_pol_2.15:= FALSE;
	
	// per
	vsState_KP_per.0:= run_tflap_noria_10210 OR run_tflap_scalp_10210;
	vsState_KP_per.1:= run_tflap_bunk_20001_10710 OR run_tflap_bunk_20002_10710;
	vsState_KP_per.2:= run_tflap_bunk_20003_10720 OR run_tflap_bunk_20004_10720;
	vsState_KP_per.3:= run_tflap_bunk_20005_10730 OR run_tflap_bunk_20006_10730;
	vsState_KP_per.4:= run_tflap_bunk_20007_10740 OR run_tflap_bunk_20008_10740;
	vsState_KP_per.5:= FALSE;
	vsState_KP_per.6:= FALSE;
	vsState_KP_per.7:= FALSE;
	vsState_KP_per.8:= FALSE;
	vsState_KP_per.9:= FALSE;
	vsState_KP_per.10:= FALSE;
	vsState_KP_per.11:= FALSE;
	vsState_KP_per.12:= FALSE;
	vsState_KP_per.13:= FALSE;
	vsState_KP_per.14:= FALSE;
	vsState_KP_per.15:= FALSE;
	
	//Alarm
	vsState_KP_DA.0:= da_tflap_10210;
	vsState_KP_DA.1:= da_tflap_10710;
	vsState_KP_DA.2:= da_tflap_10720;
	vsState_KP_DA.3:= da_tflap_10730;
	vsState_KP_DA.4:= da_tflap_10740;
	vsState_KP_DA.5:= FALSE;
	vsState_KP_DA.6:= FALSE;
	vsState_KP_DA.7:= FALSE;
	vsState_KP_DA.8:= FALSE;
	vsState_KP_DA.9:= FALSE;
	vsState_KP_DA.10:= FALSE;
	vsState_KP_DA.11:= FALSE;
	vsState_KP_DA.12:= FALSE;
	vsState_KP_DA.13:= FALSE;
	vsState_KP_DA.14:= FALSE;
	vsState_KP_DA.15:= FALSE;
	
// Задвижки
	// Открыт
	vsState_Z_opened.0:= opened_sh_10610;
	vsState_Z_opened.1:= opened_sh_10620;
	vsState_Z_opened.2:= opened_sh_10630;
	vsState_Z_opened.3:= opened_sh_10640;
	vsState_Z_opened.4:= opened_sh_30110;
	vsState_Z_opened.5:= opened_sh_21310;
	vsState_Z_opened.6:= opened_sh_21320;
	vsState_Z_opened.7:= opened_sh_21330;
	vsState_Z_opened.8:= opened_sh_30910;
	vsState_Z_opened.9:= opened_sh_30920;
	vsState_Z_opened.10:= opened_sh_30930;
	vsState_Z_opened.11:= opened_sh_30940;
	vsState_Z_opened.12:= opened_sh_30820;
	vsState_Z_opened.13:= opened_sh_30810;
	vsState_Z_opened.14:= FALSE;
	vsState_Z_opened.15:= FALSE;
	
	// Закрыт
	vsState_Z_closed.0:= closed_sh_10610;
	vsState_Z_closed.1:= closed_sh_10620;
	vsState_Z_closed.2:= closed_sh_10630;
	vsState_Z_closed.3:= closed_sh_10640;
	vsState_Z_closed.4:= closed_sh_30110;
	vsState_Z_closed.5:= closed_sh_21310;
	vsState_Z_closed.6:= closed_sh_21320;
	vsState_Z_closed.7:= closed_sh_21330;
	vsState_Z_closed.8:= closed_sh_30910;
	vsState_Z_closed.9:= closed_sh_30920;
	vsState_Z_closed.10:= closed_sh_30930;
	vsState_Z_closed.11:= closed_sh_30940;
	vsState_Z_closed.12:= closed_sh_30820;
	vsState_Z_closed.13:= closed_sh_30810;
	vsState_Z_closed.14:= FALSE;
	vsState_Z_closed.15:= FALSE;
	
	// Переключение
	vsState_Z_per.0:= NOT opened_sh_10610 AND NOT closed_sh_10610;
	vsState_Z_per.1:= NOT opened_sh_10620 AND NOT closed_sh_10620;
	vsState_Z_per.2:= NOT opened_sh_10630 AND NOT closed_sh_10630;
	vsState_Z_per.3:= NOT opened_sh_10640 AND NOT closed_sh_10640;
	vsState_Z_per.4:= NOT opened_sh_30110 AND NOT closed_sh_30110;
	vsState_Z_per.5:= NOT opened_sh_21310 AND NOT closed_sh_21310;
	vsState_Z_per.6:= NOT opened_sh_21320 AND NOT closed_sh_21320;
	vsState_Z_per.7:= NOT opened_sh_21330 AND NOT closed_sh_21330;
	vsState_Z_per.8:= NOT opened_sh_30910 AND NOT closed_sh_30910;
	vsState_Z_per.9:= NOT opened_sh_30920 AND NOT closed_sh_30920;
	vsState_Z_per.10:= NOT opened_sh_30930 AND NOT closed_sh_30930;
	vsState_Z_per.11:= NOT opened_sh_30940 AND NOT closed_sh_30940;
	vsState_Z_per.12:= NOT opened_sh_30820 AND NOT closed_sh_30820;
	vsState_Z_per.13:= NOT opened_sh_30810 AND NOT closed_sh_30810;
	vsState_Z_per.14:= FALSE;
	vsState_Z_per.15:= FALSE;
	
	// Авария
	vsState_Z_DA.0:= da_sh_10610;
	vsState_Z_DA.1:= da_sh_10620;
	vsState_Z_DA.2:= da_sh_10630;
	vsState_Z_DA.3:= da_sh_10640;
	vsState_Z_DA.4:= da_sh_30110;
	vsState_Z_DA.5:= da_sh_21310;
	vsState_Z_DA.6:= da_sh_21320;
	vsState_Z_DA.7:= da_sh_21330;
	vsState_Z_DA.8:= da_sh_30910;
	vsState_Z_DA.9:= da_sh_30920;
	vsState_Z_DA.10:= da_sh_30930;
	vsState_Z_DA.11:= da_sh_30940;
	vsState_Z_DA.12:= da_sh_30820;
	vsState_Z_DA.13:= da_sh_30810;
	vsState_Z_DA.14:= FALSE;
	vsState_Z_DA.15:= FALSE;
	
// Подсветка линий на окне загрузка сырья
	vsState_Line_load_K.0:= run_noria_10200;
	vsState_Line_load_K.1:= run_noria_10200 AND stPoz_scalp_10210;
	vsState_Line_load_K.2:= run_noria_10200 AND stPoz_noria_10210;
	vsState_Line_load_K.3:= run_scalp AND run_pch_scalp;
	vsState_Line_load_K.4:= run_noria_10400;
	vsState_Line_load_K.5:= run_sktr_10500 AND opened_sh_10610 AND stPoz_bunk1_10710;
	vsState_Line_load_K.6:= run_sktr_10500 AND opened_sh_10610 AND stPoz_bunk2_10710;
	vsState_Line_load_K.7:= run_sktr_10500 AND opened_sh_10620 AND stPoz_bunk3_10720;
	vsState_Line_load_K.8:= run_sktr_10500 AND opened_sh_10620 AND stPoz_bunk4_10720;
	vsState_Line_load_K.9:= run_sktr_10500 AND opened_sh_10630 AND stPoz_bunk5_10730;
	vsState_Line_load_K.10:= run_sktr_10500 AND opened_sh_10630 AND stPoz_bunk6_10730;
	vsState_Line_load_K.11:= run_sktr_10500 AND opened_sh_10640 AND stPoz_bunk7_10740;
	vsState_Line_load_K.12:= run_sktr_10500 AND opened_sh_10640 AND stPoz_bunk8_10740;
	vsState_Line_load_K.13:= run_noria_21200;
	vsState_Line_load_K.14:= run_shnek_21300 AND opened_sh_21310;
	vsState_Line_load_K.15:= run_shnek_21300 AND opened_sh_21320;
	
	vsState_Line_load_K1.0:= run_shnek_21300 AND opened_sh_21330;;
	vsState_Line_load_K1.1:= run_shnek_21300 AND NOT opened_sh_21310 AND NOT opened_sh_21320 AND NOT opened_sh_21330;
	vsState_Line_load_K1.2:= run_noria_30700;
	vsState_Line_load_K1.3:= run_sktr_30900 AND opened_sh_30940;
	vsState_Line_load_K1.4:= run_sktr_30900 AND opened_sh_30930;
	vsState_Line_load_K1.5:= run_sktr_30900 AND opened_sh_30920;
	vsState_Line_load_K1.6:= run_sktr_30900 AND opened_sh_30910;
	vsState_Line_load_K1.7:= run_sktr_30800 AND opened_sh_30820;
	vsState_Line_load_K1.8:= run_sktr_30800 AND opened_sh_30810;
	vsState_Line_load_K1.9:= run_shnek_30640 AND run_pch_sktr_30640;
	vsState_Line_load_K1.10:= run_sktr_20110;
	vsState_Line_load_K1.11:= run_noria_20300;
	vsState_Line_load_K1.12:= run_pch_30200;
	vsState_Line_load_K1.13:= run_pch_30200;
	vsState_Line_load_K1.14:= run_shnek_30330 AND run_pch_sktr_30330;
	vsState_Line_load_K1.15:= run_shnek_21600;
	
	vsState_Line_load_K2.0:= run_noria_30500;
	vsState_Line_load_K2.1:= run_sktr_30900 AND NOT opened_sh_30910 AND NOT opened_sh_30920 AND NOT opened_sh_30930 AND NOT opened_sh_30940;
	vsState_Line_load_K2.2:= FALSE;
	vsState_Line_load_K2.3:= FALSE;
	vsState_Line_load_K2.4:= FALSE;
	vsState_Line_load_K2.5:= FALSE;
	vsState_Line_load_K2.6:= FALSE;
	vsState_Line_load_K2.7:= FALSE;
	vsState_Line_load_K2.8:= FALSE;
	vsState_Line_load_K2.9:= FALSE;
	vsState_Line_load_K2.10:= FALSE;
	vsState_Line_load_K2.11:= FALSE;
	vsState_Line_load_K2.12:= FALSE;
	vsState_Line_load_K2.13:= FALSE;
	vsState_Line_load_K2.14:= FALSE;
	vsState_Line_load_K2.15:= FALSE;
	
// Отображение аварийных стопов на экране
	vsState_emer.0:= localstop_sktr_10110 OR localstop_end_sktr_10110;
	vsState_emer.1:= localstop_but_noria_10200 OR localstop_top_noria_10200;
	vsState_emer.2:= localstop_but_noria_10400 OR localstop_top_noria_10400;
	vsState_emer.3:= localstop_sktr_10500 OR localstop_end_sktr_10500;
	vsState_emer.4:= localstop_sktr_20110 OR localstop_end_sktr_20110;
	vsState_emer.5:= localstop_but_noria_20300 OR localstop_top_noria_20300;
	vsState_emer.6:= localstop_but_noria_21200 OR localstop_top_noria_21200;
	vsState_emer.7:= localstop_shnek_21300;
	vsState_emer.8:= localstop_shnek_30330;
	vsState_emer.9:= localstop_sktr_30400 OR localstop_end_sktr_30400;
	vsState_emer.10:= localstop_but_noria_30500 OR localstop_top_noria_30500;
	vsState_emer.11:= localstop_shnek30640;
	vsState_emer.12:= localstop_but_noria_30700 OR localstop_top_noria_30700;
	vsState_emer.13:= localstop_sktr_30900 OR localstop_end_sktr_30900;
	vsState_emer.14:= localstop_sktr_30800 OR localstop_end_sktr_30800;
	vsState_emer.15:= localstop_21600;
	
	vsState_emer1.0:= localstop_doz_shnek_20011;
	vsState_emer1.1:= localstop_doz_shnek_20012;
	vsState_emer1.2:= localstop_doz_shnek_20013;
	vsState_emer1.3:= localstop_doz_shnek_20014;
	vsState_emer1.4:= localstop_doz_shnek_20015;
	vsState_emer1.5:= localstop_doz_shnek_20016;
	vsState_emer1.6:= localstop_doz_shnek_20017;
	vsState_emer1.7:= localstop_doz_shnek_20018;
	vsState_emer1.8:= localstop_doz_shnek_21510;
	vsState_emer1.9:= localstop_doz_shnek_21520;
	vsState_emer1.10:= localstop_doz_shnek_21530;
	vsState_emer1.11:= localstop_doz_shnek_21540;
	vsState_emer1.12:= localstop_doz_shnek_21405;
	vsState_emer1.13:= localstop_doz_shnek_21406;
	vsState_emer1.14:= localstop_doz_shnek_21407;
	vsState_emer1.15:= localstop_doz_shnek_21408;
	
	vsState_emer2.0:= localstop_doz_shnek_21409;
	vsState_emer2.1:= localstop_fan_hole;
	vsState_emer2.2:= FALSE;
	vsState_emer2.3:= FALSE;
	vsState_emer2.4:= FALSE;
	vsState_emer2.5:= FALSE;
	vsState_emer2.6:= FALSE;
	vsState_emer2.7:= FALSE;
	vsState_emer2.8:= FALSE;
	vsState_emer2.9:= FALSE;
	vsState_emer2.10:= FALSE;
	vsState_emer2.11:= FALSE;
	vsState_emer2.12:= FALSE;
	vsState_emer2.13:= FALSE;
	vsState_emer2.14:= FALSE;
	vsState_emer2.15:= FALSE;

END_PROGRAM

// PLC_241/Application/FB/ASP/shluz
FUNCTION_BLOCK shluz
VAR_INPUT
	erraz: BOOL;
	dks: BOOL;
	timeDKS: TIME;
	timeStart: TIME;
	timeStop: TIME;
	next: BOOL;
	prev: BOOL;
	conditionToWork: BOOL;
	ressetErrors: BOOL;
	g_emer: BOOL;
	m_hand: BOOL;
	m_naladka: BOOL;
	hand: BOOL;
	offdks: BOOL;
	
END_VAR
VAR_OUTPUT
	run: BOOL;
	rr: BOOL;
	da: BOOL;
	errDKS: BOOL;
	resHand: BOOL;
END_VAR
VAR
	TON_DKS_OFF: TON;
	TON_DKS_ON: TON;
	TON_START: TON;
	start: BOOL;
	TON_STOP: TON;
END_VAR
VAR // added by the converter: edge detectors and wires of the graphical bodies
    _w1 : BOOL;
END_VAR

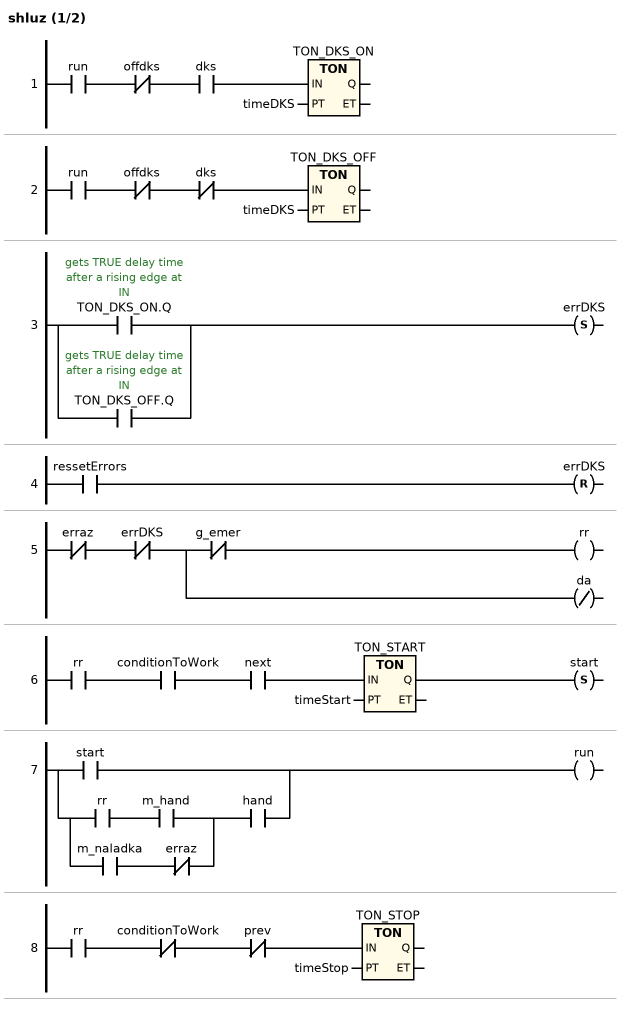
// NETWORK 1
TON_DKS_ON(IN := run AND NOT offdks AND dks, PT := timeDKS); // TON

// NETWORK 2
TON_DKS_OFF(IN := run AND NOT offdks AND NOT dks, PT := timeDKS); // TON

// NETWORK 3
//   TON_DKS_ON.Q: gets TRUE delay time after a rising edge at IN
//   TON_DKS_OFF.Q: gets TRUE delay time after a rising edge at IN
errDKS S= TON_DKS_ON.Q OR TON_DKS_OFF.Q;

// NETWORK 4
errDKS R= ressetErrors;

// NETWORK 5
_w1 := NOT erraz AND NOT errDKS;
rr := _w1 AND NOT g_emer;
da := NOT _w1;

// NETWORK 6
TON_START(IN := rr AND conditionToWork AND next, PT := timeStart); // TON
start S= TON_START.Q;

// NETWORK 7
run := start OR (rr AND m_hand OR m_naladka AND NOT erraz) AND hand;

// NETWORK 8
TON_STOP(IN := rr AND NOT conditionToWork AND NOT prev, PT := timeStop); // TON

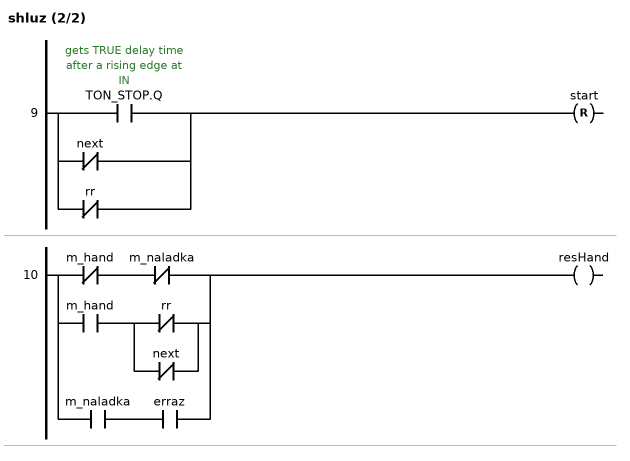
// NETWORK 9
//   TON_STOP.Q: gets TRUE delay time after a rising edge at IN
start R= TON_STOP.Q OR NOT next OR NOT rr;

// NETWORK 10
resHand := NOT m_hand AND NOT m_naladka OR m_hand AND (NOT rr OR NOT next) OR m_naladka AND erraz;

END_FUNCTION_BLOCK

// PLC_241/Application/FB/vibr/VB
FUNCTION_BLOCK VB
VAR_INPUT
	erraz: BOOL;
	timeStart: TIME;
	timeStop: TIME;
	next: BOOL;
	prev: BOOL;
	conditionToWork: BOOL;
	g_emer: BOOL;
	m_hand: BOOL;
	m_naladka: BOOL;
	hand: BOOL;
	
END_VAR
VAR_OUTPUT
	run: BOOL;
	rr: BOOL;
	da: BOOL;
	resHand: BOOL;
	
END_VAR
VAR
	TON_START: TON;
	start: BOOL;
	TON_STOP: TON;
	preb: BOOL;
END_VAR
VAR // added by the converter: edge detectors and wires of the graphical bodies
    _w1 : BOOL;
END_VAR

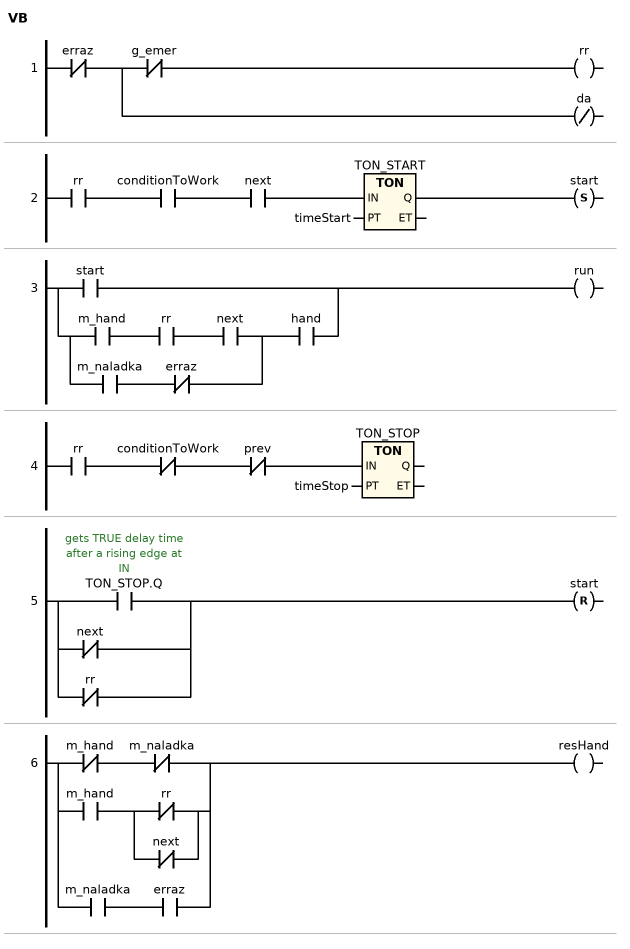
// NETWORK 1
_w1 := NOT erraz;
rr := _w1 AND NOT g_emer;
da := NOT _w1;

// NETWORK 2
TON_START(IN := rr AND conditionToWork AND next, PT := timeStart); // TON
start S= TON_START.Q;

// NETWORK 3
run := start OR (m_hand AND rr AND next OR m_naladka AND NOT erraz) AND hand;

// NETWORK 4
TON_STOP(IN := rr AND NOT conditionToWork AND NOT prev, PT := timeStop); // TON

// NETWORK 5
//   TON_STOP.Q: gets TRUE delay time after a rising edge at IN
start R= TON_STOP.Q OR NOT next OR NOT rr;

// NETWORK 6
resHand := NOT m_hand AND NOT m_naladka OR m_hand AND (NOT rr OR NOT next) OR m_naladka AND erraz;

END_FUNCTION_BLOCK
